DATA_BLOCK "DB3323"
TITLE =	TITLE ==CH2++ZNE02_Alarm_List
{ S7_language := '16(1) Italiano (Italia)  10.08.2015  13:02:09' }
VERSION : 0.1


  STRUCT
   CM_ID : STRING  [8 ] := '=CH2_2';	//IDENTIFICATIVO TRATTO
   STATION_ID : STRING  [8 ] := '++ZNE02';	//TRATTO - ZONA - STAZIONE
   ELEMENT_ID : STRING  [8 ];	//ELEMENTO
   DB_ID : INT  := 3;	//GRANDEZZA DB O TIPO
   PART_IDENTIFICATION : STRING  [12 ];	//IDENTIFICAZIONE PEZZO IN LAVORAZIONE
   ACT_CYCLE_TIME : INT ;	//TEMPO CICLO EFFETTIVO
   COUNT_GOOD : INT ;	//PEZZO PRODOTTO BUONO
   COUNT_SCRAP : INT ;	//PEZZO PRODOTTO DI SCARTO
   ACCUMULATORS : ARRAY  [0 .. 15 ] OF //ACCUMULI
   INT ;
   SPARE_01 : ARRAY  [0 .. 17 ] OF //RISERVE
   INT ;
   CODE_EVENT : ARRAY  [0 .. 7 ] OF //CODICI DI DIAGNOSTICA (codici a 4 cifre)
   INT ;
   EVENTS : STRUCT 	//EVENTI DI DIAGNOSTICA / MONITORAGGIO (bit)
    E0001 : BOOL ;	//=CH2_2++ZNE02+HCZ01-DMC01;FALHA NO MÓDULO ET200S;1
    E0002 : BOOL ;	//=CH2_2++ZNE02+HCZ01-DSW01;FALHA DE SCALANCE;1
    E0003 : BOOL ;	//=CH2_2++ZNE02+HCZ01-QF_06;ALIMENTAÇÃO MAGNETOTÉRMICA PARA CIRCUITOS AUXILIARES;1
    E0004 : BOOL ;	//=CH2_2++ZNE02+HCZ01-QF_07;POTÊNCIA MAGNETOTÉRMICA. COMANDOS E SINAIS DE SAÍDA;1
    E0005 : BOOL ;	//=CH2_2++ZNE02+HCZ01-QF_08;MAGNETOTHERM.;1
    E0006 : BOOL ;	//=CH2_2++ZNE02+HCZ01-QF_09;POTÊNCIA MAGNETOTÉRMICA. MÓDULOS E SWITCHES E/S ET200;1
    E0007 : BOOL ;
    E0008 : BOOL ;
    E0009 : BOOL ;	//=CH2_2++ZNE02+HKL02-SQ_04;MANIPULADORES DIREITOS COMPACTOS;1
    E0010 : BOOL ;	//=CH2_2++ZNE02+HKL02-SQ_10;MANIPULADORES ESQUERDOS EM TAMANHO COMPACTO;1
    E0011 : BOOL ;
    E0012 : BOOL ;
    E0013 : BOOL ;
    E0014 : BOOL ;
    E0015 : BOOL ;
    E0016 : BOOL ;
    E0017 : BOOL ;	//=CH2_2++ZNE02+HCZ01-QF_25;GRUPO DE ROTAÇÃO DA FONTE DE ALIMENTAÇÃO 440Vac +CR_01;1
    E0018 : BOOL ;	//=CH2_2++ZNE02+HCZ01-QF_26;PODER GRUPO DE ROTAÇÃO DE BACKUP 440Vac +CR_01;1
    E0019 : BOOL ;	//=CH2_2++ZNE02+HCZ01-QF_27;GRUPO DE ROTAÇÃO DA FONTE DE ALIMENTAÇÃO 440Vac +CR_02;1
    E0020 : BOOL ;	//=CH2_2++ZNE02+HCZ01-QF_28;PODER GRUPO DE ROTAÇÃO DE BACKUP 440Vac +CR_02;1
    E0021 : BOOL ;	//=CH2_2++ZNE02+HCZ01-QF_29;FONTE DE ALIMENTAÇÃO 440Vac CADEIA+TC_01;1
    E0022 : BOOL ;	//=CH2_2++ZNE02+HCZ01-QF_30;MAGNETOTHERM.440Vac FREIO GR.ROTAÇÃO +CR_01;1
    E0023 : BOOL ;	//=CH2_2++ZNE02+HCZ01-QF_31;MAGNETOTHERM.440Vac FREIO GR.ROTAÇÃO BK +CR_01;1
    E0024 : BOOL ;	//=CH2_2++ZNE02+HCZ01-QF_32;MAGNETOTHERM.440Vac FREIO GR.ROTAÇÃO +CR_02;1
    E0025 : BOOL ;	//=CH2_2++ZNE02+HCZ01-QF_33;MAGNETOTHERM.440Vac FREIO GR.ROTAÇÃO BK +CR_02;1
    E0026 : BOOL ;	//=CH2_2++ZNE02+HCZ01-QF_34;MAGNETOTERM.440Vac FREIO DE CORRENTE +TC_01;1
    E0027 : BOOL ;	//=CH2_2++ZNE02+HCZ01-QF_35;MAGNETOTERM.440Vac CADEIA DE BACKUP +TC_01;1
    E0028 : BOOL ;	//=CH2_2++ZNE02+HCZ01-QF_36;MAGNETOTERM.440Vac FREIO DE CORRENTE DE BACKUP +TC_01;1
    E0029 : BOOL ;	//=CH2_2++ZNE02+HCZ01-BT_01;SOBRETEMPERATURA DO RESISTOR DE FRENAGEM +CR_01;1
    E0030 : BOOL ;	//=CH2_2++ZNE02+HCZ01-BT_02;SOBRETEMP DO RESISTOR DE FRENAGEM DE BACKUP.;1
    E0031 : BOOL ;	//=CH2_2++ZNE02+HCZ01-BT_03;SOBRETEMPERATURA DO RESISTOR DE FRENAGEM +CR_02;1
    E0032 : BOOL ;	//=CH2_2++ZNE02+HCZ01-BT_04;SOBRETEMP DO RESISTOR DE FRENAGEM DE BACKUP.;1
    E0033 : BOOL ;	//=CH2_2++ZNE02+HCZ01-U__01;FALHA MOVIDRIVE +CR_01;1
    E0034 : BOOL ;	//=CH2_2++ZNE02+HCZ01-U__02;FALHA DE BACKUP DO MOVIDRIVE +CR_01;1
    E0035 : BOOL ;	//=CH2_2++ZNE02+HCZ01-U__03;FALHA MOVIDRIVE +CR_02;1
    E0036 : BOOL ;	//=CH2_2++ZNE02+HCZ01-U__04;FALHA DE BACKUP DO MOVIDRIVE +CR_02;1
    E0037 : BOOL ;	//=CH2_2++ZNE02+HCZ01-U__05;FALHA MOVIDRIVE +TC_01;1
    E0038 : BOOL ;	//=CH2_2++ZNE02+HCZ01-U__06;FALHA DE BACKUP DO MOVIDRIVE +TC_01;1
    E0039 : BOOL ;	//=CH2_2++ZNE02+HCZ01-U__01;MOVIDRIVE +CR_01 ERRO DE COMUNICAÇÃO;1
    E0040 : BOOL ;	//=CH2_2++ZNE02+HCZ01-U__02;ERRO DE COMUNICAÇÃO BACKUP DO MOVIDRIVE +CR_01;1
    E0041 : BOOL ;	//=CH2_2++ZNE02+HCZ01-U__03;MOVIDRIVE +CR_02 ERRO DE COMUNICAÇÃO;1
    E0042 : BOOL ;	//=CH2_2++ZNE02+HCZ01-U__04;ERRO DE COMUNICAÇÃO BACKUP DO MOVIDRIVE +CR_02;1
    E0043 : BOOL ;	//=CH2_2++ZNE02+HCZ01-U__05;MOVIDRIVE +TC_01 ERRO DE COMUNICAÇÃO;1
    E0044 : BOOL ;	//=CH2_2++ZNE02+HCZ01-U__06;ERRO COMUNICADO. BACKUP DO MOVIDRIVE +TC_01;1
    E0045 : BOOL ;	//=CH2_2++ZNE02+HCZ01-KMS02;EFICIÊNCIA DO RELÉ 440Vac SET_2 +CR_01;1
    E0046 : BOOL ;	//=CH2_2++ZNE02+HCZ01-KMS04;EFICIÊNCIA DO RELÉ 440Vca SET_4 +CR_02;1
    E0047 : BOOL ;	//=CH2_2++ZNE02+HCZ01-KMS06;EFICIÊNCIA DO RELÉ 440Vac SET_5 +TC_01;1
    E0048 : BOOL ;	//=CH2_2++ZNE02+HCZ01-KAS02;CONJUNTO DE EFICIÊNCIA DO RELÉ 24Vdc_2 +CR_01;1
    E0049 : BOOL ;	//=CH2_2++ZNE02+HCZ01-KAS04;CONJUNTO DE EFICIÊNCIA DO RELÉ 24Vdc_4 +CR_02;1
    E0050 : BOOL ;	//=CH2_2++ZNE02+HCZ01-KAS06;CONJUNTO DE EFICIÊNCIA DO RELÉ 24Vdc_5 +TC_01;1
    E0051 : BOOL ;	//=CH2_2++ZNE02+PTZ01-DMC01;FALHA NO MÓDULO ET200S;1
    E0052 : BOOL ;	//=CH2_2++ZNE02+PTZ02-DMC01;FALHA NO MÓDULO ET200S;1
    E0053 : BOOL ;	//=CH2_2++ZNE02+HKL01-DMC01;FALHA NO MÓDULO ET200S;1
    E0054 : BOOL ;	//=CH2_2++ZNE02+HKL02-DMC01;FALHA NO MÓDULO ET200S;1
    E0055 : BOOL ;	//=CH2_2++ZNE02+XGA01-SC_01;PORTÃO EM ANOMALIA;1
    E0056 : BOOL ;	//=CH2_2++ZNE02+XGA02-SC_01;PORTÃO EM ANOMALIA;1
    E0057 : BOOL ;	//=CH2_2++ZNE02+XGA05-SC_01;PORTÃO EM ANOMALIA;1
    E0058 : BOOL ;	//=CH2_2++ZNE02+XGA06-SC_01;PORTÃO EM ANOMALIA;1
    E0059 : BOOL ;
    E0060 : BOOL ;
    E0061 : BOOL ;
    E0062 : BOOL ;
    E0063 : BOOL ;
    E0064 : BOOL ;
    E0065 : BOOL ;	//=CH2_2++ZNE02+HCZ01-DMC01;ANOMALIA DO MÓDULO ProfSafe ET200S-FDI-FDO;2
    E0066 : BOOL ;	//=CH2_2++ZNE02+PTZ01-DMC01;ANOMALIA DO MÓDULO ProfSafe ET200S-FDI;2
    E0067 : BOOL ;	//=CH2_2++ZNE02+PTZ02-DMC01;ANOMALIA DO MÓDULO ProfSafe ET200S-FDI;2
    E0068 : BOOL ;	//=CH2_2++ZNE02+PTZ03-DMC01;ANOMALIA DO MÓDULO ProfSafe ET200S-FDI;2
    E0069 : BOOL ;	//=CH2_2++ZNE02+PRE01-DMC01;ANOMALIA DO MÓDULO ProfSafe ET200S-FDI;2
    E0070 : BOOL ;	//=CH2_2++ZNE02+HKL01-DMC01;ANOMALIA DO MÓDULO ProfSafe ET200S-FDI;2
    E0071 : BOOL ;	//=CH2_2++ZNE02+HKL02-DMC01;ANOMALIA DO MÓDULO ProfSafe ET200S-FDI;2
    E0072 : BOOL ;
    E0073 : BOOL ;
    E0074 : BOOL ;
    E0075 : BOOL ;
    E0076 : BOOL ;
    E0077 : BOOL ;	//=CH2_2++ZNE02+XGA06-SC_01;MANUTENÇÃO PROGRAMADA DE ACESSO ABERTO (PM);13
    E0078 : BOOL ;	//=CH2_2++ZNE02+XGA06-SC_01;LIMPEZA TÉCNICA DE ACESSO ABERTO (AM);14
    E0079 : BOOL ;	//=CH2_2++ZNE02+XGA06-SC_01;ACESSO NÃO RESTAURADO MANUTENÇÃO DO PROGRAMA (PM);13
    E0080 : BOOL ;	//=CH2_2++ZNE02+XGA06-SC_01;ACESSO NÃO RESTAURADO LIMPEZA TÉCNICA (AM);14
    E0081 : BOOL ;	//=CH2_2++ZNE02+PTZ01-SB_07;BOTÃO DE EMERGENCIA APERTADO;2
    E0082 : BOOL ;	//=CH2_2++ZNE02+PTZ01-SB_07;EMERGÊNCIA NÃO RESTAURADA;2
    E0083 : BOOL ;	//=CH2_2++ZNE02+PTZ02-SB_07;BOTÃO DE EMERGENCIA APERTADO;2
    E0084 : BOOL ;	//=CH2_2++ZNE02+PTZ02-SB_07;EMERGÊNCIA NÃO RESTAURADA;2
    E0085 : BOOL ;	//=CH2_2++ZNE02+PGA01-SB_01;BOTÃO DE EMERGENCIA APERTADO;2
    E0086 : BOOL ;	//=CH2_2++ZNE02+PGA01-SB_01;EMERGÊNCIA NÃO RESTAURADA;2
    E0087 : BOOL ;	//=CH2_2++ZNE02+PGA02-SB_01;BOTÃO DE EMERGENCIA APERTADO;2
    E0088 : BOOL ;	//=CH2_2++ZNE02+PGA02-SB_01;EMERGÊNCIA NÃO RESTAURADA;2
    E0089 : BOOL ;	//=CH2_2++ZNE02+SLL01-SB_01;CORDA DE EMERGÊNCIA DO LADO ESQUERDO PUXADA;2
    E0090 : BOOL ;	//=CH2_2++ZNE02+SLL01-SB_01;CORDA DE EMERGÊNCIA LADO ESQUERDO NÃO RESTAURADA;2
    E0091 : BOOL ;	//=CH2_2++ZNE02+SLL02-SB_01;CORDA DE EMERGÊNCIA DO LADO DIREITO PUXADA;2
    E0092 : BOOL ;	//=CH2_2++ZNE02+SLL02-SB_01;CORDA DE EMERGÊNCIA LADO DIREITO NÃO RESTAURADA;2
    E0093 : BOOL ;	//=CH2_2++ZNE02+SLL03-SB_01;CORDA DE EMERGÊNCIA DO LADO ESQUERDO PUXADA;2
    E0094 : BOOL ;	//=CH2_2++ZNE02+SLL03-SB_01;CORDA DE EMERGÊNCIA LADO ESQUERDO NÃO RESTAURADA;2
    E0095 : BOOL ;	//=CH2_2++ZNE02+SLL04-SB_01;CORDA DE EMERGÊNCIA DO LADO DIREITO PUXADA;2
    E0096 : BOOL ;	//=CH2_2++ZNE02+SLL04-SB_01;CORDA DE EMERGÊNCIA LADO DIREITO NÃO RESTAURADA;2
    E0097 : BOOL ;	//=CH2_2++ZNE02+SLL05-SB_01;CORDA DE EMERGÊNCIA DO LADO ESQUERDO PUXADA;2
    E0098 : BOOL ;	//=CH2_2++ZNE02+SLL05-SB_01;CORDA DE EMERGÊNCIA LADO ESQUERDO NÃO RESTAURADA;2
    E0099 : BOOL ;	//=CH2_2++ZNE02+SLL06-SB_01;CORDA DE EMERGÊNCIA DO LADO DIREITO PUXADA;2
    E0100 : BOOL ;	//=CH2_2++ZNE02+SLL06-SB_01;CORDA DE EMERGÊNCIA LADO DIREITO NÃO RESTAURADA;2
    E0101 : BOOL ;	//=CH2_2++ZNE02+XGA01-SC_01;ACESSO ABERTO NÃO PROGRAMADO (GM);2
    E0102 : BOOL ;	//=CH2_2++ZNE02+XGA01-SC_01;ACESSO NÃO RESTAURADO(GM);2
    E0103 : BOOL ;	//=CH2_2++ZNE02+XGA02-SC_01;ACESSO ABERTO NÃO PROGRAMADO (GM);2
    E0104 : BOOL ;	//=CH2_2++ZNE02+XGA02-SC_01;ACESSO NÃO RESTAURADO(GM);2
    E0105 : BOOL ;	//=CH2_2++ZNE02+XGA05-SC_01;ACESSO ABERTO NÃO PROGRAMADO (GM);2
    E0106 : BOOL ;	//=CH2_2++ZNE02+XGA05-SC_01;ACESSO NÃO RESTAURADO(GM);2
    E0107 : BOOL ;	//=CH2_2++ZNE02+XGA06-SC_01;ACESSO ABERTO NÃO PROGRAMADO (GM);2
    E0108 : BOOL ;	//=CH2_2++ZNE02+XGA06-SC_01;ACESSO NÃO RESTAURADO(GM);2
    E0109 : BOOL ;	//=CH2_2++ZNE02+PRB01-VT_01;BARREIRA ATIVADA (ESTAÇÃO 77);2
    E0110 : BOOL ;	//=CH2_2++ZNE02+PRB01-VT_01;BARREIRA NÃO RESTAURADA (ESTAÇÃO 77);2
    E0111 : BOOL ;	//=CH2_2++ZNE02+PRB02-VT_02;BARREIRA ATIVADA (ESTAÇÃO 78);2
    E0112 : BOOL ;	//=CH2_2++ZNE02+PRB02-VT_02;BARREIRA NÃO RESTAURADA (ESTAÇÃO 78);2
    E0113 : BOOL ;	//=CH2_2++ZNE02+PRB03-VT_03;BARREIRA ATIVADA (ESTAÇÃO Q2);2
    E0114 : BOOL ;	//=CH2_2++ZNE02+PRB03-VT_03;BARREIRA NÃO RESTAURADA (ESTAÇÃO Q2);2
    E0115 : BOOL ;	//=CH2_2++ZNE02+PRB04-VT_04;BARREIRA ATIVADA (ESTAÇÃO Q3);2
    E0116 : BOOL ;	//=CH2_2++ZNE02+PRB04-VT_04;BARREIRA NÃO RESTAURADA (ESTAÇÃO Q3);2
    E0117 : BOOL ;	//=CH2_2++ZNE02+XGA01-SC_01;MANUTENÇÃO PROGRAMADA DE ACESSO ABERTO (PM);13
    E0118 : BOOL ;	//=CH2_2++ZNE02+XGA01-SC_01;LIMPEZA TÉCNICA DE ACESSO ABERTO (AM);14
    E0119 : BOOL ;	//=CH2_2++ZNE02+XGA01-SC_01;ACESSO NÃO RESTAURADO PROG. DE MANUTENÇÃO (PM);13
    E0120 : BOOL ;	//=CH2_2++ZNE02+XGA01-SC_01;ACESSO NÃO RESTAURADO LIMPEZA TÉCNICA (AM);14
    E0121 : BOOL ;	//=CH2_2++ZNE02+XGA02-SC_01;MANUTENÇÃO PROGRAMADA DE ACESSO ABERTO (PM);13
    E0122 : BOOL ;	//=CH2_2++ZNE02+XGA02-SC_01;LIMPEZA TÉCNICA DE ACESSO ABERTO (AM);14
    E0123 : BOOL ;	//=CH2_2++ZNE02+XGA02-SC_01;ACESSO NÃO RESTAURADO PROG. DE MANUTENÇÃO (PM);13
    E0124 : BOOL ;	//=CH2_2++ZNE02+XGA02-SC_01;ACESSO NÃO RESTAURADO LIMPEZA TÉCNICA (AM);14
    E0125 : BOOL ;	//=CH2_2++ZNE02+XGA05-SC_01;MANUTENÇÃO PROGRAMADA DE ACESSO ABERTO (PM);13
    E0126 : BOOL ;	//=CH2_2++ZNE02+XGA05-SC_01;LIMPEZA TÉCNICA DE ACESSO ABERTO (AM);14
    E0127 : BOOL ;	//=CH2_2++ZNE02+XGA05-SC_01;ACESSO NÃO RESTAURADO PROG. DE MANUTENÇÃO (PM);13
    E0128 : BOOL ;	//=CH2_2++ZNE02+XGA05-SC_01;ACESSO NÃO RESTAURADO LIMPEZA TÉCNICA (AM);14
    E0129 : BOOL ;	//=CH2_2++ZNE02+HCZ01-QF_03;FONTE DE ALIMENTAÇÃO MAGNETOTÉRMICA PARA AR CONDICIONADO 400V;58
    E0130 : BOOL ;	//=CH2_2++ZNE02+HCZ01-QF_15;MAGNETO. PODER PAINEL OPERADOR 24Vdc +PTZ01;58
    E0131 : BOOL ;	//=CH2_2++ZNE02+HCZ01-QF_16;MAGNETO. PODER PAINEL OPERADOR 24Vdc +PTZ02;58
    E0132 : BOOL ;	//=CH2_2++ZNE02+HCZ01-U__01;PRÉ-ALARME MOVIDRIVE +CR_01;58
    E0133 : BOOL ;	//=CH2_2++ZNE02+HCZ01-U__02;PRÉ-ALARME DE BACKUP DO MOVIDRIVE +CR_01;58
    E0134 : BOOL ;	//=CH2_2++ZNE02+HCZ01-U__03;PRÉ-ALARME MOVIDRIVE +CR_02;58
    E0135 : BOOL ;	//=CH2_2++ZNE02+HCZ01-U__04;PRÉ-ALARME DE BACKUP DO MOVIDRIVE +CR_02;58
    E0136 : BOOL ;	//=CH2_2++ZNE02+HCZ01-U__05;PRÉ-ALARME MOVIDRIVE +TC_01;58
    E0137 : BOOL ;	//=CH2_2++ZNE02+HCZ01-U__06;PRÉ-ALARME DE BACKUP DO MOVIDRIVE +TC_01;58
    E0138 : BOOL ;	//=CH2_2++ZNE02+PTZ01-DSP01;PRÉ-ALARME SEM PLC <-> COMUNICAÇÃO IHM;58
    E0139 : BOOL ;	//=CH2_2++ZNE02+PTZ02-DSP01;PRÉ-ALARME SEM PLC <-> COMUNICAÇÃO IHM;58
    E0140 : BOOL ;	//=CH2_2++ZNE02+PTZ01-SA_03;PEDIDO DE ACESSO PARA MANUTENÇÃO PLANEJADA (PM);58
    E0141 : BOOL ;	//=CH2_2++ZNE02+PTZ01-SA_03;SOLICITAR ACESSO PARA LIMPEZA TÉCNICA (AM);58
    E0142 : BOOL ;	//=CH2_2++ZNE02+PTZ02-SA_03;PEDIDO DE ACESSO PARA MANUTENÇÃO PLANEJADA (PM);58
    E0143 : BOOL ;	//=CH2_2++ZNE02+PTZ02-SA_03;SOLICITAR ACESSO PARA LIMPEZA TÉCNICA (AM);58
    E0144 : BOOL ;	//=CH2_2++ZNE02+PGA01-SA_01;PEDIDO DE ACESSO PARA MANUTENÇÃO PLANEJADA (PM);58
    E0145 : BOOL ;	//=CH2_2++ZNE02+PGA01-SA_01;SOLICITAR ACESSO PARA LIMPEZA TÉCNICA (AM);58
    E0146 : BOOL ;	//=CH2_2++ZNE02+PGA02-SA_01;PEDIDO DE ACESSO PARA MANUTENÇÃO PLANEJADA (PM);58
    E0147 : BOOL ;	//=CH2_2++ZNE02+PGA02-SA_01;SOLICITAR ACESSO PARA LIMPEZA TÉCNICA (AM);58
    E0148 : BOOL ;	//=CH2_2++ZNE02+PTZ01-SA_03;SOLICITAR ACESSO PARA MANUTENÇÃO NÃO PROGRAMADA (GM);58
    E0149 : BOOL ;	//=CH2_2++ZNE02+PTZ02-SA_03;SOLICITAR ACESSO PARA MANUTENÇÃO NÃO PROGRAMADA (GM);58
    E0150 : BOOL ;	//=CH2_2++ZNE02+PGA01-SA_01;SOLICITAR ACESSO PARA MANUTENÇÃO NÃO PROGRAMADA (GM);58
    E0151 : BOOL ;	//=CH2_2++ZNE02+PGA02-SA_01;SOLICITAR ACESSO PARA MANUTENÇÃO NÃO PROGRAMADA (GM);58
    E0152 : BOOL ;	//=CH2_2++ZNE02+HCZ01-ST_01;CONTROLE DE TEMPERATURA DO GABINETE;58
    E0153 : BOOL ;	//=CH2_2++ZNE02+HAU01-QF_01;ALIMENTAÇÃO TÉRMICA 440Vac USUÁRIOS NO LADO DA LINHA;58
    E0154 : BOOL ;	//=CH2_2++ZNE02+HAU01-QF_02;PARAFUSO 220Vac TORX T50 PARA FIXAÇÃO. FIVELA DIREITA;58
    E0155 : BOOL ;	//=CH2_2++ZNE02+HAU01-QF_03;PARAFUSO FIXO TÉRMICO 220Vac. BANCO TRASEIRO =CH2++ZNE0;58
    E0156 : BOOL ;	//=CH2_2++ZNE02+HAU01-QF_04;ESTRUTURA TÉRMICA 220Vac FIX INFERIOR DIREITA =CH2++ZNE;58
    E0157 : BOOL ;	//=CH2_2++ZNE02+HAU01-QF_05;ÂNCORA/TUBO 220Vac. ESCAPE =CH2++ZNE02+FRM;58
    E0158 : BOOL ;	//=CH2_2++ZNE02+HAU01-QF_06;220Vac TORX T50 PARA FIXAÇÃO DE FILIAL ESQUERDO FIVELA =CH2++ZNE;58
    E0159 : BOOL ;	//=CH2_2++ZNE02+HAU01-QF_07;220Vac FIX SUPORTE INFERIOR ESQUERDO =CH2++ZNE02+FRM06;58
    E0160 : BOOL ;	//=CH2_2++ZNE02+HAU01-QF_08;ALIMENTAÇÃO TÉRMICA 220Vac USUÁRIO 7;58
    E0161 : BOOL ;	//=CH2_2++ZNE02+HAU01-QF_09;ALIMENTAÇÃO TÉRMICA 220Vac USUÁRIO 8;58
    E0162 : BOOL ;	//=CH2_2++ZNE02+HAU01-QF_10;ALIMENTAÇÃO TÉRMICA 220Vac USUÁRIO 9;58
    E0163 : BOOL ;	//=CH2_2++ZNE02+HCZ01;PRÉ-ALARME DE SEGURANÇA DE BYPASS ATIVO;54
    E0164 : BOOL ;
    E0165 : BOOL ;
    E0166 : BOOL ;
    E0167 : BOOL ;
    E0168 : BOOL ;
    E0169 : BOOL ;	//=CH2_2++ZNE02+HAU02-QF_01;ALIMENTAÇÃO TÉRMICA 440Vac USUÁRIOS NO LADO DA LINHA;58
    E0170 : BOOL ;	//=CH2_2++ZNE02+HAU02-QF_02;CRISTAIS 220Vac (CARGA) =CH2++ZNE02+PTN01;58
    E0171 : BOOL ;	//=CH2_2++ZNE02+HAU02-QF_03;PÁRA-BRISA 220Vac B.U - LINHA =CH2++ZNE02+FRM04;58
    E0172 : BOOL ;	//=CH2_2++ZNE02+HAU02-QF_04;ALIMENTAÇÃO TÉRMICA 220Vac USUÁRIO 3;58
    E0173 : BOOL ;	//=CH2_2++ZNE02+HAU02-QF_05;ALIMENTAÇÃO TÉRMICA 220Vac USUÁRIO 4;58
    E0174 : BOOL ;	//=CH2_2++ZNE02+HAU02-QF_06;ALIMENTAÇÃO TÉRMICA 220Vac USUÁRIO 5;58
    E0175 : BOOL ;	//=CH2_2++ZNE02+HAU02-QF_07;ALIMENTAÇÃO TÉRMICA 220Vac USUÁRIO 6;58
    E0176 : BOOL ;	//=CH2_2++ZNE02+HAU02-QF_08;ALIMENTAÇÃO TÉRMICA 220Vac USUÁRIO 7;58
    E0177 : BOOL ;	//=CH2_2++ZNE02+HAU02-QF_09;ALIMENTAÇÃO TÉRMICA 220Vac USUÁRIO 8;58
    E0178 : BOOL ;	//=CH2_2++ZNE02+HAU02-QF_10;ALIMENTAÇÃO TÉRMICA 220Vac USUÁRIO 9;58
    E0179 : BOOL ;
    E0180 : BOOL ;
    E0181 : BOOL ;
    E0182 : BOOL ;
    E0183 : BOOL ;
    E0184 : BOOL ;
    E0185 : BOOL ;	//=CH2_2++ZNE02+HAU03-QF_01;ALIMENTAÇÃO TÉRMICA 440Vac USUÁRIOS NO LADO DA LINHA;58
    E0186 : BOOL ;	//=CH2_2++ZNE02+HAU03-QF_02;ALIMENTAÇÃO TÉRMICA 220Vac USUÁRIO 1;58
    E0187 : BOOL ;	//=CH2_2++ZNE02+HAU03-QF_03;ALIMENTAÇÃO TÉRMICA 220Vac USUÁRIO 2;58
    E0188 : BOOL ;	//=CH2_2++ZNE02+HAU03-QF_04;ALIMENTAÇÃO TÉRMICA 220Vac USUÁRIO 3;58
    E0189 : BOOL ;	//=CH2_2++ZNE02+HAU03-QF_05;ALIMENTAÇÃO TÉRMICA 220Vac USUÁRIO 4;58
    E0190 : BOOL ;	//=CH2_2++ZNE02+HAU03-QF_06;ALIMENTAÇÃO TÉRMICA 220Vac USUÁRIO 5;58
    E0191 : BOOL ;	//=CH2_2++ZNE02+HAU03-QF_07;ALIMENTAÇÃO TÉRMICA 220Vac USUÁRIO 6;58
    E0192 : BOOL ;	//=CH2_2++ZNE02+HAU03-QF_08;ALIMENTAÇÃO TÉRMICA 220Vac USUÁRIO 7;58
    E0193 : BOOL ;	//=CH2_2++ZNE02+HAU03-QF_09;ALIMENTAÇÃO TÉRMICA 220Vac USUÁRIO 8;58
    E0194 : BOOL ;	//=CH2_2++ZNE02+HAU03-QF_10;ALIMENTAÇÃO TÉRMICA 220Vac USUÁRIO 9;58
    E0195 : BOOL ;
    E0196 : BOOL ;
    E0197 : BOOL ;
    E0198 : BOOL ;
    E0199 : BOOL ;
    E0200 : BOOL ;
    E0201 : BOOL ;	//=CH2_2++ZNE02+PTZ01;SETOR ASCENTE NÃO ESTÁ EM CICLO INICIADO;58
    E0202 : BOOL ;	//=CH2_2++ZNE02+PTZ01;SETOR JUSANTE NÃO ESTÁ EM CICLO INICIADO;58
    E0203 : BOOL ;	//=CH2_2++ZNE02+PTZ02;SETOR ASCENTE NÃO ESTÁ EM CICLO INICIADO;58
    E0204 : BOOL ;	//=CH2_2++ZNE02+PTZ02;SETOR JUSANTE NÃO ESTÁ EM CICLO INICIADO;58
    E0205 : BOOL ;	//=CH2_2++ZNE02+PTZ03;SETOR ASCENTE NÃO ESTÁ EM CICLO INICIADO;58
    E0206 : BOOL ;	//=CH2_2++ZNE02+PTZ03;SETOR JUSANTE NÃO ESTÁ EM CICLO INICIADO;58
    E0207 : BOOL ;	//=CH2_2++ZNE02+PRE01;SETOR ASCENTE NÃO ESTÁ EM CICLO INICIADO;58
    E0208 : BOOL ;	//=CH2_2++ZNE02+PRE01;SETOR JUSANTE NÃO ESTÁ EM CICLO INICIADO;58
    E0209 : BOOL ;	//=CH2_2++ZNE02;EM PRODUÇÃO;19
    E0210 : BOOL ;	//=CH2_2++ZNE02+PTZ01-SB_05;INICIAR CICLO AUTOMÁTICO;15
    E0211 : BOOL ;	//=CH2_2++ZNE02+PTZ02-SB_05;INICIAR CICLO AUTOMÁTICO;15
    E0212 : BOOL ;	//=CH2_2++ZNE02+PTZ01-SA_01;CICLO MANUAL SELECIONADO;16
    E0213 : BOOL ;	//=CH2_2++ZNE02+PTZ02-SA_01;CICLO MANUAL SELECIONADO;16
    E0214 : BOOL ;	//=CH2_2++ZNE02+PTZ01-SB_04;PARADA DO CICLO;17
    E0215 : BOOL ;	//=CH2_2++ZNE02+PTZ02-SB_04;PARADA DO CICLO;17
    E0216 : BOOL ;
    E0217 : BOOL ;
    E0218 : BOOL ;
    E0219 : BOOL ;
    E0220 : BOOL ;
    E0221 : BOOL ;
    E0222 : BOOL ;
    E0223 : BOOL ;
    E0224 : BOOL ;
    E0225 : BOOL ;	//=CH2_2++ZNE02+TC_01-SQ_04;FC FALHA DENTE PARADA TEMPORÁRIA SEM GANCHO;1
    E0226 : BOOL ;	//=CH2_2++ZNE02+TC_01-SQ_05;FC FALHA DENTE PARADA TEMPORÁRIA SEM GANCHO;1
    E0227 : BOOL ;
    E0228 : BOOL ;
    E0229 : BOOL ;
    E0230 : BOOL ;	//=CH2_2++ZNE02+TC_01-SQ_06;CONTROLE ANTI-VARA DE CADEIA;1
    E0231 : BOOL ;
    E0232 : BOOL ;
    E0233 : BOOL ;	//=CH2_2++ZNE02+TC_01-SE_01;CONTROLE DE ROTAÇÃO DA CADEIA;1
    E0234 : BOOL ;	//=CH2_2++ZNE02+TC_01-B__01;VERIFICAÇÃO DE CADEIA LENTA;1
    E0235 : BOOL ;	//=CH2_2++ZNE02+TC_01-SE_01;FALHA DO CODIFICADOR WIP;1
    E0236 : BOOL ;
    E0237 : BOOL ;	//=CH2_2++ZNE02+TC_01;CTRL EXECUTAR TTS ENTRADA DO CHASSIS;1
    E0238 : BOOL ;	//=CH2_2++ZNE02+TC_01;CTRL RUN TTS SAÍDA DO CHASSIS;1
    E0239 : BOOL ;
    E0240 : BOOL ;
    E0241 : BOOL ;	//=CH2_2++ZNE02+TC_01;PARCEIRO 1 NÃO FORA DO LADO ESQUERDO;10
    E0242 : BOOL ;	//=CH2_2++ZNE02+TC_01;PARCEIRO 2 NÃO FORA DAS DIMENSÕES DO LADO DIREITO;10
    E0243 : BOOL ;	//=CH2_2++ZNE02+TC_01;PARCEIRO 3 NÃO FORA DO LADO ESQUERDO;10
    E0244 : BOOL ;	//=CH2_2++ZNE02+TC_01;PARCEIRO 4 NÃO FORA DAS DIMENSÕES DO LADO DIREITO;10
    E0245 : BOOL ;	//=CH2_2++ZNE02+TC_01;PARCEIRO 5 NÃO FORA DO LADO ESQUERDO;10
    E0246 : BOOL ;	//=CH2_2++ZNE02+TC_01;PARCEIRO 6 NÃO FORA DAS DIMENSÕES DO LADO DIREITO;10
    E0247 : BOOL ;	//=CH2_2++ZNE02+TC_01;PARCEIRO 7 NÃO FORA DO LADO ESQUERDO;10
    E0248 : BOOL ;	//=CH2_2++ZNE02+TC_01;PARCEIRO 8 NÃO FORA DAS DIMENSÕES DO LADO DIREITO;10
    E0249 : BOOL ;	//=CH2_2++ZNE02+TC_01;PRÉ-ALARME DE BYPASS DE FALHA ATIVO;58
    E0250 : BOOL ;	//=CH2_2++ZNE02+TC_01;FALTA PRÉ-ALARME DE HABILITAÇÃO MECÂNICA;58
    E0251 : BOOL ;
    E0252 : BOOL ;
    E0253 : BOOL ;
    E0254 : BOOL ;
    E0255 : BOOL ;
    E0256 : BOOL ;
    E0257 : BOOL ;	//=CH2_2++ZNE02+TC_01;FALHA NO CARREGAMENTO;6
    E0258 : BOOL ;	//=CH2_2++ZNE02+TC_01;FALHA NO DESCARREGAMENTO;9
    E0259 : BOOL ;
    E0260 : BOOL ;
    E0261 : BOOL ;
    E0262 : BOOL ;
    E0263 : BOOL ;
    E0264 : BOOL ;
    E0265 : BOOL ;	//=CH2_2++ZNE02+TC_01;ESVAZIAMENTO EM ANDAMENTO;58
    E0266 : BOOL ;
    E0267 : BOOL ;
    E0268 : BOOL ;
    E0269 : BOOL ;
    E0270 : BOOL ;
    E0271 : BOOL ;
    E0272 : BOOL ;
    E0273 : BOOL ;	//=CH2_2++ZNE02+CR_01-SQ_01;VERIFIQUE A QUEBRA DA CORRENTE DIREITA;1
    E0274 : BOOL ;	//=CH2_2++ZNE02+CR_01-SQ_02;VERIFIQUE A QUEBRA DA CORRENTE ESQUERDA;1
    E0275 : BOOL ;	//=CH2_2++ZNE02+CR_01-SQ_03;VERIFICAÇÃO DO BLOCO DE SEGURANÇA DO GANCHO DE FALHA FC;1
    E0276 : BOOL ;
    E0277 : BOOL ;	//=CH2_2++ZNE02+CR_01-SQ_05;CONTROLE DE POSIÇÃO DE REPOUSO DE FALHA FC;1
    E0278 : BOOL ;	//=CH2_2++ZNE02+CR_01-SQ_06;Obturador desengatado;1
    E0279 : BOOL ;	//=CH2_2++ZNE02+CR_01-SQ_07;FC FALHA INÍCIO DE ROTAÇÃO DO GANCHO;1
    E0280 : BOOL ;	//=CH2_2++ZNE02+CR_01-SQ_08;CONTROLE DE POSIÇÃO DE FALHA FC NO TRABALHO;1
    E0281 : BOOL ;	//=CH2_2++ZNE02+CR_01-SQ_09;FALHA DO FC FORA DO ESPAÇO;1
    E0282 : BOOL ;	//=CH2_2++ZNE02+CR_01-SQE01;EXTRACURSO GR. ROTAÇÃO DE DESCANSO;1
    E0283 : BOOL ;	//=CH2_2++ZNE02+CR_01-SQE02;EXTRACURSO GR. ROTAÇÃO DE TRABALHO;1
    E0284 : BOOL ;	//=CH2_2++ZNE02+CR_01-SQA01;FC FALHA ROTAÇÃO DO GANCHO PARADA DESCANSO;1
    E0285 : BOOL ;	//=CH2_2++ZNE02+CR_01-SQA02;FC FAULT STOP TRABALHO DE ROTAÇÃO DO GANCHO;1
    E0286 : BOOL ;	//=CH2_2++ZNE02+CR_01-SQS01;FC FALHA ROTAÇÃO DO GANCHO LENTA;1
    E0287 : BOOL ;	//=CH2_2++ZNE02+CR_01-SQS02;FALHA FC DESACELERAÇÃO DA ROTAÇÃO DO GANCHO DE TRABALHO;1
    E0288 : BOOL ;	//=CH2_2++ZNE02+CR_01-SQ_10;FC FALHA PRESENÇA DA RODA CAM DO OBTURADOR;1
    E0289 : BOOL ;	//=CH2_2++ZNE02+CR_01-SQ_04;CONTROLE DE BLOQUEIO DE ROTAÇÃO;1
    E0290 : BOOL ;	//=CH2_2++ZNE02+CR_01-SQA01;TEMPO DE ROTAÇÃO DO GANCHO EM REPOUSO;1
    E0291 : BOOL ;	//=CH2_2++ZNE02+CR_01-SQA02;TEMPO DE ROTAÇÃO DO GANCHO NO TRABALHO;1
    E0292 : BOOL ;	//=CH2_2++ZNE02+CR_01;FORA DA ETAPA_00;1
    E0293 : BOOL ;	//=CH2_2++ZNE02+CR_01;FORA DA ETAPA_05;1
    E0294 : BOOL ;	//=CH2_2++ZNE02+CR_01;FORA DA ETAPA_10;1
    E0295 : BOOL ;	//=CH2_2++ZNE02+CR_01;FORA DA ETAPA_15;1
    E0296 : BOOL ;	//=CH2_2++ZNE02+CR_01;FALHA NA ROTAÇÃO DO GANCHO;1
    E0297 : BOOL ;	//=CH2_2++ZNE02+CR_01;ANOMALIA DE SELEÇÃO DE LINHA/BACKUP MOVIDRIVE;1
    E0298 : BOOL ;	//=CH2_2++ZNE02+CR_01-M__01;ALARME DE CORRENTE ABSORVIDA;1
    E0299 : BOOL ;
    E0300 : BOOL ;
    E0301 : BOOL ;
    E0302 : BOOL ;
    E0303 : BOOL ;
    E0304 : BOOL ;
    E0305 : BOOL ;	//=CH2_2++ZNE02+CR_01;PRÉ-ALARME DE CORRENTE SOLTA;58
    E0306 : BOOL ;
    E0307 : BOOL ;
    E0308 : BOOL ;
    E0309 : BOOL ;
    E0310 : BOOL ;
    E0311 : BOOL ;
    E0312 : BOOL ;
    E0313 : BOOL ;	//=CH2_2++ZNE02+CR_01;PRÉ-ALARME DE BYPASS DE FALHA ATIVO;58
    E0314 : BOOL ;
    E0315 : BOOL ;
    E0316 : BOOL ;
    E0317 : BOOL ;
    E0318 : BOOL ;
    E0319 : BOOL ;
    E0320 : BOOL ;
    E0321 : BOOL ;
    E0322 : BOOL ;
    E0323 : BOOL ;
    E0324 : BOOL ;
    E0325 : BOOL ;
    E0326 : BOOL ;
    E0327 : BOOL ;
    E0328 : BOOL ;
    E0329 : BOOL ;	//=CH2_2++ZNE02+CR_01;CICLO AUTOMÁTICO PASSO A PASSO INICIADO;58
    E0330 : BOOL ;
    E0331 : BOOL ;
    E0332 : BOOL ;
    E0333 : BOOL ;
    E0334 : BOOL ;
    E0335 : BOOL ;
    E0336 : BOOL ;
    E0337 : BOOL ;	//=CH2_2++ZNE02+CR_02-SQ_01;VERIFIQUE A QUEBRA DA CORRENTE DIREITA;1
    E0338 : BOOL ;	//=CH2_2++ZNE02+CR_02-SQ_02;VERIFIQUE A QUEBRA DA CORRENTE ESQUERDA;1
    E0339 : BOOL ;	//=CH2_2++ZNE02+CR_02-SQ_03;VERIFICAÇÃO DO BLOCO DE SEGURANÇA DO GANCHO DE FALHA FC;1
    E0340 : BOOL ;
    E0341 : BOOL ;	//=CH2_2++ZNE02+CR_02-SQ_05;CONTROLE DE POSIÇÃO DE REPOUSO DE FALHA FC;1
    E0342 : BOOL ;	//=CH2_2++ZNE02+CR_02-SQ_06;Obturador desengatado;1
    E0343 : BOOL ;	//=CH2_2++ZNE02+CR_02-SQ_07;FC FALHA INÍCIO DE ROTAÇÃO DO GANCHO;1
    E0344 : BOOL ;	//=CH2_2++ZNE02+CR_02-SQ_08;CONTROLE DE POSIÇÃO DE FALHA FC NO TRABALHO;1
    E0345 : BOOL ;	//=CH2_2++ZNE02+CR_02-SQ_09;FALHA DO FC FORA DO ESPAÇO;1
    E0346 : BOOL ;	//=CH2_2++ZNE02+CR_02-SQE01;EXTRACURSO GR. ROTAÇÃO DE DESCANSO;1
    E0347 : BOOL ;	//=CH2_2++ZNE02+CR_02-SQE02;EXTRACURSO GR. ROTAÇÃO DE TRABALHO;1
    E0348 : BOOL ;	//=CH2_2++ZNE02+CR_02-SQA01;FC FALHA ROTAÇÃO DO GANCHO PARADA DESCANSO;1
    E0349 : BOOL ;	//=CH2_2++ZNE02+CR_02-SQA02;FC FAULT STOP TRABALHO DE ROTAÇÃO DO GANCHO;1
    E0350 : BOOL ;	//=CH2_2++ZNE02+CR_02-SQS01;FC FALHA ROTAÇÃO DO GANCHO LENTA;1
    E0351 : BOOL ;	//=CH2_2++ZNE02+CR_02-SQS02;FALHA FC DESACELERAÇÃO DA ROTAÇÃO DO GANCHO DE TRABALHO;1
    E0352 : BOOL ;	//=CH2_2++ZNE02+CR_02-SQ_10;FC FALHA PRESENÇA DA RODA CAM DO OBTURADOR;1
    E0353 : BOOL ;	//=CH2_2++ZNE02+CR_02-SQ_04;CONTROLE DE BLOQUEIO DE ROTAÇÃO;1
    E0354 : BOOL ;	//=CH2_2++ZNE02+CR_02-SQA01;TEMPO DE ROTAÇÃO DO GANCHO EM REPOUSO;1
    E0355 : BOOL ;	//=CH2_2++ZNE02+CR_02-SQA02;TEMPO DE ROTAÇÃO DO GANCHO NO TRABALHO;1
    E0356 : BOOL ;	//=CH2_2++ZNE02+CR_02;FORA DA ETAPA_00;1
    E0357 : BOOL ;	//=CH2_2++ZNE02+CR_02;FORA DA ETAPA_05;1
    E0358 : BOOL ;	//=CH2_2++ZNE02+CR_02;FORA DA ETAPA_10;1
    E0359 : BOOL ;	//=CH2_2++ZNE02+CR_02;FORA DA ETAPA_15;1
    E0360 : BOOL ;	//=CH2_2++ZNE02+CR_02;FALHA NA ROTAÇÃO DO GANCHO;1
    E0361 : BOOL ;	//=CH2_2++ZNE02+CR_02;ANOMALIA DE SELEÇÃO DE LINHA/BACKUP MOVIDRIVE;1
    E0362 : BOOL ;	//=CH2_2++ZNE02+CR_02-M__01;ALARME DE CORRENTE ABSORVIDA;1
    E0363 : BOOL ;
    E0364 : BOOL ;
    E0365 : BOOL ;
    E0366 : BOOL ;
    E0367 : BOOL ;
    E0368 : BOOL ;
    E0369 : BOOL ;	//=CH2_2++ZNE02+CR_02;PRÉ-ALARME DE CORRENTE SOLTA;58
    E0370 : BOOL ;
    E0371 : BOOL ;
    E0372 : BOOL ;
    E0373 : BOOL ;
    E0374 : BOOL ;
    E0375 : BOOL ;
    E0376 : BOOL ;
    E0377 : BOOL ;	//=CH2_2++ZNE02+CR_02;PRÉ-ALARME DE BYPASS DE FALHA ATIVO;58
    E0378 : BOOL ;
    E0379 : BOOL ;
    E0380 : BOOL ;
    E0381 : BOOL ;
    E0382 : BOOL ;
    E0383 : BOOL ;
    E0384 : BOOL ;
    E0385 : BOOL ;
    E0386 : BOOL ;
    E0387 : BOOL ;
    E0388 : BOOL ;
    E0389 : BOOL ;
    E0390 : BOOL ;
    E0391 : BOOL ;
    E0392 : BOOL ;
    E0393 : BOOL ;	//=CH2_2++ZNE02+CR_02;CICLO AUTOMÁTICO PASSO A PASSO INICIADO;58
    E0394 : BOOL ;	//=CH2_2++ZNE02+WIP01;Anomalia na leitura de código de barras/etiqueta;5
    E0395 : BOOL ;	//=CH2_2++ZNE02+WIP01;Tempo limite de leitura de código de barras/etiqueta;5
    E0396 : BOOL ;	//=CH2_2++ZNE02+WIP01;Inconsistência físico-lógica;5
    E0397 : BOOL ;	//=CH2_2++ZNE02+WIP01;Dígito de verificação CIS incorreto;5
    E0398 : BOOL ;	//=CH2_2++ZNE02+WIP01;Tempo limite de recepção de dados da rota anterior;5
    E0399 : BOOL ;	//=CH2_2++ZNE02+WIP01;Inconsistência de dados do ponto de ajuste do CIS/VIS com o CIS/VIS a seguir;5
    E0400 : BOOL ;	//=CH2_2++ZNE02+WIP01;Serviço MES Setpoint não ativo;58
    E0401 : BOOL ;	//=CH2_2++ZNE02+WIP01;Solução para desligamento de linha do MES/PLC para chamada de operadora.;11
    E0402 : BOOL ;	//=CH2_2++ZNE02+WIP01;Serviço MES Tr;10
    E0403 : BOOL ;	//=CH2_2++ZNE02+WIP01;NOK para continuar a partir da estação automática MES (SAService);10
    E0404 : BOOL ;	//=CH2_2++ZNE02+WIP01;Rota Wip do serviço MES não ativa;58
    E0405 : BOOL ;	//=CH2_2++ZNE02+WIP01;Configuração da estação de serviço MES não ativa;58
    E0406 : BOOL ;	//=CH2_2++ZNE02+WIP01;Chamada do Operador de Serviço MES;58
    E0407 : BOOL ;	//=CH2_2++ZNE02+WIP01;Serviço de estação de envio de dados MES SAService não ativo;58
    E0408 : BOOL ;	//=CH2_2++ZNE02+WIP01;Serviço de estação de solicitação de dados MES SRService não ativo;58
    E0409 : BOOL ;	//=CH2_2++ZNE02+WIP01;Serviço de modelo de estação MES SMService não ativo;58
    E0410 : BOOL ;	//=CH2_2++ZNE02+WIP01;Trate wip em modificação;17
    E0411 : BOOL ;	//=CH2_2++ZNE02+WIP01;Estação não automática;16
    E0412 : BOOL ;	//=CH2_2++ZNE02+WIP01;PARADA DE LINHA POR MÊS;17
    E0413 : BOOL ;	//=CH2_2++ZNE02+WIP01;Leitor de bypass CIS NEXT do MES;55
    E0414 : BOOL ;	//=CH2_2++ZNE02+WIP01;Estação excluída;1
    E0415 : BOOL ;	//=CH2_2++ZNE02+WIP01;Lista de estações de configuração de votação;10
    E0416 : BOOL ;
    E0417 : BOOL ;	//=CH2_2++ZNE02+LMN01-DSP01;OPERADOR CHAMADA LIMO 01 ESTAÇÃO 75 SX;53
    E0418 : BOOL ;	//=CH2_2++ZNE02+LMN03-DSP01;OPERADOR CHAMADA LIMO 03 ESTAÇÃO 76 SX;53
    E0419 : BOOL ;	//=CH2_2++ZNE02+LMN05-DSP01;OPERADOR CHAMADA LIMO 05 ESTAÇÃO 77 SX;53
    E0420 : BOOL ;	//=CH2_2++ZNE02+LMN07-DSP01;OPERADOR CHAMADA LIMO 07 ESTAÇÃO 78 SX;53
    E0421 : BOOL ;	//=CH2_2++ZNE02+LMN09-DSP01;OPERADOR CHAMADA LIMO 09 ESTAÇÃO 79 SX;53
    E0422 : BOOL ;	//=CH2_2++ZNE02+LMN11-DSP01;OPERADOR DE LIMO CHAMADA 11 ESTAÇÃO 80 SX;53
    E0423 : BOOL ;	//=CH2_2++ZNE02+LMN13-DSP01;OPERADOR CHAMADA LIMO 13 ESTAÇÃO 81 ESQUERDA;53
    E0424 : BOOL ;	//=CH2_2++ZNE02+LMN15-DSP01;CHAMADA DE OPERADOR DE LIMO 15 ESTAÇÃO Q2 ESQUERDA;53
    E0425 : BOOL ;	//=CH2_2++ZNE02+LMN17-DSP01;CHAMADA DE OPERADOR DE LIMO 17 ESTAÇÃO Q3 ESQUERDA;53
    E0426 : BOOL ;
    E0427 : BOOL ;
    E0428 : BOOL ;
    E0429 : BOOL ;
    E0430 : BOOL ;
    E0431 : BOOL ;
    E0432 : BOOL ;
    E0433 : BOOL ;	//=CH2_2++ZNE02+LMN02-DSP01;OPERADOR CHAMADA LIMO 02 ESTAÇÃO 75 DX;53
    E0434 : BOOL ;	//=CH2_2++ZNE02+LMN04-DSP01;OPERADOR CHAMADA LIMO 04 ESTAÇÃO 76 DX;53
    E0435 : BOOL ;	//=CH2_2++ZNE02+LMN06-DSP01;OPERADOR CHAMADA LIMO 06 ESTAÇÃO 77 DX;53
    E0436 : BOOL ;	//=CH2_2++ZNE02+LMN08-DSP01;OPERADOR CHAMADA LIMO 08 ESTAÇÃO 78 DX;53
    E0437 : BOOL ;	//=CH2_2++ZNE02+LMN10-DSP01;CHAMADA DE OPERADOR LIMO 10 ESTAÇÃO 79 DX;53
    E0438 : BOOL ;	//=CH2_2++ZNE02+LMN12-DSP01;CHAMADA DE OPERADOR LIMO 12 ESTAÇÃO 80 DX;53
    E0439 : BOOL ;	//=CH2_2++ZNE02+LMN14-DSP01;CHAMADA DE OPERADOR LIMO 14 ESTAÇÃO 81 DX;53
    E0440 : BOOL ;	//=CH2_2++ZNE02+LMN16-DSP01;CHAMADA DE OPERADOR DE LIMO 16 ESTAÇÃO Q2 DX;53
    E0441 : BOOL ;	//=CH2_2++ZNE02+LMN18-DSP01;CHAMADA DE OPERADOR DE LIMO 18 ESTAÇÃO Q3 DX;53
    E0442 : BOOL ;
    E0443 : BOOL ;
    E0444 : BOOL ;
    E0445 : BOOL ;
    E0446 : BOOL ;
    E0447 : BOOL ;
    E0448 : BOOL ;
    E0449 : BOOL ;	//=CH2_2++ZNE02+LMN01-DSP01;PARADA LATERAL DO SILT LINE 01 ESTAÇÃO 75 ESQUERDA;12
    E0450 : BOOL ;	//=CH2_2++ZNE02+LMN03-DSP01;PARADA LATERAL DO SILT LINE 03 ESTAÇÃO 76 ESQUERDA;12
    E0451 : BOOL ;	//=CH2_2++ZNE02+LMN05-DSP01;PARADA LATERAL DO SILT LINE 05 ESTAÇÃO 77 ESQUERDA;12
    E0452 : BOOL ;	//=CH2_2++ZNE02+LMN07-DSP01;PARADA LATERAL DO SILT LINE 07 ESTAÇÃO 78 ESQUERDA;12
    E0453 : BOOL ;	//=CH2_2++ZNE02+LMN09-DSP01;PARADA LADO DA LINHA DE LODO 09 ESTAÇÃO 79 ESQUERDA;12
    E0454 : BOOL ;	//=CH2_2++ZNE02+LMN11-DSP01;PARADA LADO DA LINHA DE SILT 11 ESTAÇÃO 80 ESQUERDA;12
    E0455 : BOOL ;	//=CH2_2++ZNE02+LMN13-DSP01;PARADA LADO DA LINHA DE LODO 13 ESTAÇÃO 81 ESQUERDA;12
    E0456 : BOOL ;	//=CH2_2++ZNE02+LMN15-DSP01;PARADA LATERAL DA LINHA DE SILT 15 ESTAÇÃO Q2 ESQUERDA;12
    E0457 : BOOL ;	//=CH2_2++ZNE02+LMN17-DSP01;PARADA LATERAL DO SILT LINE 17 ESTAÇÃO Q3 ESQUERDA;12
    E0458 : BOOL ;
    E0459 : BOOL ;
    E0460 : BOOL ;
    E0461 : BOOL ;
    E0462 : BOOL ;
    E0463 : BOOL ;
    E0464 : BOOL ;
    E0465 : BOOL ;	//=CH2_2++ZNE02+LMN02-DSP01;PARADA LADO DA LINHA DE LODO 02 ESTAÇÃO 75 DIREITA;12
    E0466 : BOOL ;	//=CH2_2++ZNE02+LMN04-DSP01;PARADA LADO DA LINHA DE LODO 04 ESTAÇÃO 76 DIREITA;12
    E0467 : BOOL ;	//=CH2_2++ZNE02+LMN06-DSP01;PARADA LADO DA LINHA DE LODO 06 ESTAÇÃO 77 DIREITA;12
    E0468 : BOOL ;	//=CH2_2++ZNE02+LMN08-DSP01;PARADA LADO DA LINHA DE SILT 08 ESTAÇÃO 78 DIREITA;12
    E0469 : BOOL ;	//=CH2_2++ZNE02+LMN10-DSP01;PARADA LADO DA LINHA DE SILT 10 ESTAÇÃO 79 DIREITA;12
    E0470 : BOOL ;	//=CH2_2++ZNE02+LMN12-DSP01;PARADA LADO DA LINHA DE SILT 12 ESTAÇÃO 80 DIREITA;12
    E0471 : BOOL ;	//=CH2_2++ZNE02+LMN14-DSP01;PARADA LADO DA LINHA DE SILT 14 ESTAÇÃO 81 DIREITA;12
    E0472 : BOOL ;	//=CH2_2++ZNE02+LMN16-DSP01;PARADA LADO DA LINHA DE SILT 16 ESTAÇÃO Q2 DIREITA;12
    E0473 : BOOL ;	//=CH2_2++ZNE02+LMN18-DSP01;PARADA LADO DA LINHA DE SILT 18 ESTAÇÃO Q3 DIREITA;12
    E0474 : BOOL ;
    E0475 : BOOL ;
    E0476 : BOOL ;
    E0477 : BOOL ;
    E0478 : BOOL ;
    E0479 : BOOL ;
    E0480 : BOOL ;
    E0481 : BOOL ;	//=CH2_2++ZNE02+LMN01-DSP01;LINHA PARADA OPERADOR DE LIMO 01 ESTAÇÃO 75 SX;11
    E0482 : BOOL ;	//=CH2_2++ZNE02+LMN03-DSP01;STOP OPERADOR DE LINHA LIMO 03 ESTAÇÃO 76 SX;11
    E0483 : BOOL ;	//=CH2_2++ZNE02+LMN05-DSP01;STOP OPERADOR DE LINHA LIMO 05 ESTAÇÃO 77 SX;11
    E0484 : BOOL ;	//=CH2_2++ZNE02+LMN07-DSP01;PARAR OPERADOR DE LINHA LIMO 07 ESTAÇÃO 78 SX;11
    E0485 : BOOL ;	//=CH2_2++ZNE02+LMN09-DSP01;PARAR OPERADOR DE LINHA LIMO 09 ESTAÇÃO 79 SX;11
    E0486 : BOOL ;	//=CH2_2++ZNE02+LMN11-DSP01;LINE STOP OPERADOR DE LIMO 11 ESTAÇÃO 80 SX;11
    E0487 : BOOL ;	//=CH2_2++ZNE02+LMN13-DSP01;LINHA PARADA OPERADOR DE LIMO 13 ESTAÇÃO 81 ESQUERDA;11
    E0488 : BOOL ;	//=CH2_2++ZNE02+LMN15-DSP01;PARADA DA LINHA DO OPERADOR DE LIMO 15 Q2 ESTAÇÃO À ESQUERDA;11
    E0489 : BOOL ;	//=CH2_2++ZNE02+LMN17-DSP01;PARADA DA LINHA DO OPERADOR DE LIMO 17 Q3 ESTAÇÃO À ESQUERDA;11
    E0490 : BOOL ;
    E0491 : BOOL ;
    E0492 : BOOL ;
    E0493 : BOOL ;
    E0494 : BOOL ;
    E0495 : BOOL ;
    E0496 : BOOL ;
    E0497 : BOOL ;	//=CH2_2++ZNE02+LMN02-DSP01;STOP OPERADOR DE LINHA LIMO 02 ESTAÇÃO 75 DX;11
    E0498 : BOOL ;	//=CH2_2++ZNE02+LMN04-DSP01;STOP OPERADOR DE LINHA LIMO 04 ESTAÇÃO 76 DX;11
    E0499 : BOOL ;	//=CH2_2++ZNE02+LMN06-DSP01;STOP OPERADOR DE LINHA LIMO 06 ESTAÇÃO 77 DX;11
    E0500 : BOOL ;	//=CH2_2++ZNE02+LMN08-DSP01;STOP OPERADOR DE LINHA LIMO 08 ESTAÇÃO 78 DX;11
    E0501 : BOOL ;	//=CH2_2++ZNE02+LMN10-DSP01;STOP LINE OPERADOR LIMO 10 ESTAÇÃO 79 DX;11
    E0502 : BOOL ;	//=CH2_2++ZNE02+LMN12-DSP01;ESTAÇÃO DE PARADA DA LINHA DO OPERADOR LIMO 12 80 DX;11
    E0503 : BOOL ;	//=CH2_2++ZNE02+LMN14-DSP01;PARAR OPERADOR DE LINHA LIMO 14 ESTAÇÃO 81 DX;11
    E0504 : BOOL ;	//=CH2_2++ZNE02+LMN16-DSP01;PARADA DA LINHA DO OPERADOR DE LIMO 16 Q2 ESTAÇÃO DIREITA;11
    E0505 : BOOL ;	//=CH2_2++ZNE02+LMN18-DSP01;PARADA DA LINHA DO OPERADOR DE LIMO 18 Q3 ESTAÇÃO DIREITA;11
    E0506 : BOOL ;
    E0507 : BOOL ;
    E0508 : BOOL ;
    E0509 : BOOL ;
    E0510 : BOOL ;
    E0511 : BOOL ;
    E0512 : BOOL ;
    E0513 : BOOL ;	//=CH2_2++ZNE02+HCZ02-DMC01;FALHA NO MÓDULO ET200S;1
    E0514 : BOOL ;	//=CH2_2++ZNE02+HCZ02-DSW01;FALHA DE SCALANCE;1
    E0515 : BOOL ;	//=CH2_2++ZNE02+HCZ02-QF_06;ALIMENTAÇÃO DISJUNTOR TÉRMICO PARA CIRCUITOS AUXILIARES;1
    E0516 : BOOL ;	//=CH2_2++ZNE02+HCZ02-QF_07;DISJUNTOR TÉRMICO. PODER COMANDOS E SINAIS DE SAÍDA;1
    E0517 : BOOL ;	//=CH2_2++ZNE02+HCZ02-QF_08;FONTE DE ALIMENTAÇÃO MAGNETOTÉRMICA PARA CIRCUITOS DE SEGURANÇA;1
    E0518 : BOOL ;	//=CH2_2++ZNE02+HCZ02-QF_09;DISJUNTOR TÉRMICO. PODER MÓDULOS E SWITCHES E/S ET200;1
    E0519 : BOOL ;
    E0520 : BOOL ;
    E0521 : BOOL ;
    E0522 : BOOL ;
    E0523 : BOOL ;
    E0524 : BOOL ;
    E0525 : BOOL ;
    E0526 : BOOL ;
    E0527 : BOOL ;
    E0528 : BOOL ;
    E0529 : BOOL ;	//=CH2_2++ZNE02+HCZ02-QF_10;ALIMENTAÇÃO 24Vdc MOVIFIT +TQ_01;1
    E0530 : BOOL ;	//=CH2_2++ZNE02+HCZ02-QF_20;FONTE DE ALIMENTAÇÃO 440Vac MOVIFIT +TQ_01;1
    E0531 : BOOL ;	//=CH2_2++ZNE02+HCZ02-QF_21;FONTE DE ALIMENTAÇÃO 440Vac OBTURADOR ENTRADA TTS +TQ_01;1
    E0532 : BOOL ;	//=CH2_2++ZNE02+HCZ02-QF_22;FONTE DE ALIMENTAÇÃO 440Vac SAÍDA TTS DO OBTURADOR +TQ_01;1
    E0533 : BOOL ;	//=CH2_2++ZNE02+HCZ02-QF_25;ALIMENTAÇÃO 440Vac ELEVADOR +TQ_01;1
    E0534 : BOOL ;	//=CH2_2++ZNE02+HCZ02-QF_26;FONTE DE ALIMENTAÇÃO 440Vac ELEVADOR BACKUP +TQ_01;1
    E0535 : BOOL ;	//=CH2_2++ZNE02+HCZ02-QF_27;ALIMENTAÇÃO MAGNETOTÉRMICA 440Vac TRILHA +TTS01;1
    E0536 : BOOL ;	//=CH2_2++ZNE02+HCZ02-QF_30;FONTE DE ALIMENTAÇÃO 440Vac MOTOR FREIO DO ELEVADOR +TQ_01;1
    E0537 : BOOL ;	//=CH2_2++ZNE02+HCZ02-QF_31;FREIO DO MOTOR DE BACKUP DO ELEVADOR 440Vac +TQ_01;1
    E0538 : BOOL ;	//=CH2_2++ZNE02+HCZ02-QF_32;PISTA DE FREIO DO MOTOR DE ALIMENTAÇÃO 440Vac +TTS01;1
    E0539 : BOOL ;	//=CH2_2++ZNE02+HCZ02-BT_01;SOBRETEMP. RESISTOR DE TRAVAGEM DO ELEVADOR +TQ_01;1
    E0540 : BOOL ;	//=CH2_2++ZNE02+HCZ02-BT_02;RESISTÊNCIA À FRENAGEM DO ELEVADOR DE RESERVA.;1
    E0541 : BOOL ;	//=CH2_2++ZNE02+HCZ02-U__01;FALHA MOVIDRIVE +TQ_01;1
    E0542 : BOOL ;	//=CH2_2++ZNE02+HCZ02-U__02;FALHA DE BACKUP DO MOVIDRIVE +TQ_01;1
    E0543 : BOOL ;	//=CH2_2++ZNE02+HCZ02-U__05;FALHA MOVIDRIVE +TTS01;1
    E0544 : BOOL ;	//=CH2_2++ZNE02+HCZ02-U__01;ERRO DE COMUNICAÇÃO MOVIDRIVE +TQ_01;1
    E0545 : BOOL ;	//=CH2_2++ZNE02+HCZ02-U__02;BACKUP MOVIDRIVE +TQ_01 ERRO DE COMUNICAÇÃO;1
    E0546 : BOOL ;	//=CH2_2++ZNE02+HCZ02-U__05;ERRO DE COMUNICAÇÃO MOVIDRIVE +TTS01;1
    E0547 : BOOL ;	//=CH2_2++ZNE02+HCZ02-U__01;EIXO NÃO ZERO MOVIDRIVE +TQ_01;1
    E0548 : BOOL ;	//=CH2_2++ZNE02+HCZ02-U__02;EIXO NÃO ZERO MOVIDRIVE BACKUP +TQ_01;1
    E0549 : BOOL ;	//=CH2_2++ZNE02+HCZ02-KMS02;EFICIÊNCIA DO RELÉ 440Vac +TQ_01;1
    E0550 : BOOL ;	//=CH2_2++ZNE02+HCZ02-KAS02;EFICIÊNCIA DO RELÉ 24Vdc +TQ_01;1
    E0551 : BOOL ;	//=CH2_2++ZNE02+HCZ02-KAS04;FEEDBACK 24Vdc ZONA 2 SETOR 3 TTS01;1
    E0552 : BOOL ;	//=CH2_2++ZNE02+PTZ03-DMC01;FALHA NO MÓDULO ET200S;1
    E0553 : BOOL ;	//=CH2_2++ZNE02+PRE01-DMC01;FALHA NO MÓDULO ET200S;1
    E0554 : BOOL ;	//=CH2_2++ZNE02+XGA03-SC_01;PORTÃO EM ANOMALIA;1
    E0555 : BOOL ;	//=CH2_2++ZNE02+XGA04-SC_01;PORTÃO EM ANOMALIA;1
    E0556 : BOOL ;	//=CH2_2++ZNE02+XGA06-SC_01;PORTÃO EM ANOMALIA;1
    E0557 : BOOL ;	//=CH2_2++ZNE02+XGA07-SC_01;PORTÃO EM ANOMALIA;1
    E0558 : BOOL ;	//=CH2_2++ZNE02+HCZ02-DMC01;ANOMALIA DO MÓDULO ProfSafe ET200S-FDI-FDO;2
    E0559 : BOOL ;
    E0560 : BOOL ;
    E0561 : BOOL ;
    E0562 : BOOL ;
    E0563 : BOOL ;
    E0564 : BOOL ;
    E0565 : BOOL ;
    E0566 : BOOL ;
    E0567 : BOOL ;
    E0568 : BOOL ;
    E0569 : BOOL ;
    E0570 : BOOL ;
    E0571 : BOOL ;
    E0572 : BOOL ;
    E0573 : BOOL ;
    E0574 : BOOL ;
    E0575 : BOOL ;
    E0576 : BOOL ;
    E0577 : BOOL ;
    E0578 : BOOL ;
    E0579 : BOOL ;
    E0580 : BOOL ;
    E0581 : BOOL ;
    E0582 : BOOL ;
    E0583 : BOOL ;
    E0584 : BOOL ;
    E0585 : BOOL ;
    E0586 : BOOL ;
    E0587 : BOOL ;
    E0588 : BOOL ;
    E0589 : BOOL ;
    E0590 : BOOL ;
    E0591 : BOOL ;
    E0592 : BOOL ;
    E0593 : BOOL ;	//=CH2_2++ZNE02+PTZ03-SB_07;BOTÃO DE EMERGENCIA APERTADO;2
    E0594 : BOOL ;	//=CH2_2++ZNE02+PTZ03-SB_07;EMERGÊNCIA NÃO RESTAURADA;2
    E0595 : BOOL ;	//=CH2_2++ZNE02+PRE01-SB_07;BOTÃO DE EMERGENCIA APERTADO;2
    E0596 : BOOL ;	//=CH2_2++ZNE02+PRE01-SB_07;EMERGÊNCIA NÃO RESTAURADA;2
    E0597 : BOOL ;	//=CH2_2++ZNE02+XGA03-SC_01;ACESSO ABERTO NÃO PROGRAMADO (GM);2
    E0598 : BOOL ;	//=CH2_2++ZNE02+XGA03-SC_01;ACESSO NÃO RESTAURADO(GM);2
    E0599 : BOOL ;	//=CH2_2++ZNE02+XGA04-SC_01;ACESSO ABERTO NÃO PROGRAMADO (GM);2
    E0600 : BOOL ;	//=CH2_2++ZNE02+XGA04-SC_01;ACESSO NÃO RESTAURADO(GM);2
    E0601 : BOOL ;	//=CH2_2++ZNE02+PRB05-VT_05;BARREIRA INTERDITADA;2
    E0602 : BOOL ;	//=CH2_2++ZNE02+PRB05-VT_05;BARREIRA NÃO RESTAURADA;2
    E0603 : BOOL ;	//=CH2_2++ZNE02+PGA03-SB_01;BOTÃO DE EMERGENCIA APERTADO;2
    E0604 : BOOL ;	//=CH2_2++ZNE02+PGA03-SB_01;EMERGÊNCIA NÃO RESTAURADA;2
    E0605 : BOOL ;	//=CH2_2++ZNE02+XGA07-SC_01;ACESSO ABERTO NÃO PROGRAMADO (GM);2
    E0606 : BOOL ;	//=CH2_2++ZNE02+XGA07-SC_01;ACESSO NÃO RESTAURADO(GM);2
    E0607 : BOOL ;
    E0608 : BOOL ;
    E0609 : BOOL ;
    E0610 : BOOL ;
    E0611 : BOOL ;
    E0612 : BOOL ;
    E0613 : BOOL ;
    E0614 : BOOL ;
    E0615 : BOOL ;
    E0616 : BOOL ;	//=CH2_2++ZNE02+XGA03-SC_01;ACESSO NÃO RESTAURADO LIMPEZA TÉCNICA (AM);14
    E0617 : BOOL ;	//=CH2_2++ZNE02+XGA03-SC_01;MANUTENÇÃO PROGRAMADA DE ACESSO ABERTO (PM);13
    E0618 : BOOL ;	//=CH2_2++ZNE02+XGA03-SC_01;LIMPEZA TÉCNICA DE ACESSO ABERTO (AM);14
    E0619 : BOOL ;	//=CH2_2++ZNE02+XGA03-SC_01;ACESSO NÃO RESTAURADO PROG. DE MANUTENÇÃO (PM);13
    E0620 : BOOL ;	//=CH2_2++ZNE02+XGA04-SC_01;MANUTENÇÃO PROGRAMADA DE ACESSO ABERTO (PM);13
    E0621 : BOOL ;	//=CH2_2++ZNE02+XGA04-SC_01;LIMPEZA TÉCNICA DE ACESSO ABERTO (AM);14
    E0622 : BOOL ;	//=CH2_2++ZNE02+XGA04-SC_01;ACESSO NÃO RESTAURADO PROG. DE MANUTENÇÃO (PM);13
    E0623 : BOOL ;	//=CH2_2++ZNE02+XGA07-SC_01;MANUTENÇÃO PROGRAMADA DE ACESSO ABERTO (PM);13
    E0624 : BOOL ;	//=CH2_2++ZNE02+XGA07-SC_01;LIMPEZA TÉCNICA DE ACESSO ABERTO (AM);14
    E0625 : BOOL ;	//=CH2_2++ZNE02+XGA07-SC_01;ACESSO NÃO RESTAURADO PROG. DE MANUTENÇÃO (PM);13
    E0626 : BOOL ;	//=CH2_2++ZNE02+XGA04-SC_01;ACESSO NÃO RESTAURADO LIMPEZA TÉCNICA (AM);14
    E0627 : BOOL ;	//=CH2_2++ZNE02+XGA07-SC_01;ACESSO NÃO RESTAURADO LIMPEZA TÉCNICA (AM);14
    E0628 : BOOL ;
    E0629 : BOOL ;
    E0630 : BOOL ;
    E0631 : BOOL ;
    E0632 : BOOL ;
    E0633 : BOOL ;
    E0634 : BOOL ;
    E0635 : BOOL ;
    E0636 : BOOL ;
    E0637 : BOOL ;
    E0638 : BOOL ;
    E0639 : BOOL ;
    E0640 : BOOL ;
    E0641 : BOOL ;	//=CH2_2++ZNE02+HCZ02-QF_03;FONTE DE ALIMENTAÇÃO MAGNETOTÉRMICA PARA AR CONDICIONADO 400V;58
    E0642 : BOOL ;	//=CH2_2++ZNE02+HCZ02-QF_15;MAGNETO. PODER PAINEL OPERADOR 24Vdc +PTZ03;58
    E0643 : BOOL ;	//=CH2_2++ZNE02+HCZ02-QF_16;MAGNETO. PODER PAINEL OPERADOR 24Vdc +PRE01;58
    E0644 : BOOL ;	//=CH2_2++ZNE02+HCZ02-U__01;PRÉ-ALARME MOVIDRIVE +TQ_01;58
    E0645 : BOOL ;	//=CH2_2++ZNE02+HCZ02-U__02;PRÉ-ALARME DE BACKUP DO MOVIDRIVE +TQ_01;58
    E0646 : BOOL ;	//=CH2_2++ZNE02+HCZ02-U__05;PRÉ-ALARME MOVIDRIVE +TTS01;58
    E0647 : BOOL ;	//=CH2_2++ZNE02+PTZ03-DSP01;PRÉ-ALARME SEM PLC <-> COMUNICAÇÃO IHM;58
    E0648 : BOOL ;	//=CH2_2++ZNE02+PRE01-DSP01;PRÉ-ALARME SEM PLC <-> COMUNICAÇÃO IHM;58
    E0649 : BOOL ;	//=CH2_2++ZNE02+PTZ03-SA_03;PEDIDO DE ACESSO PARA MANUTENÇÃO PLANEJADA (PM);58
    E0650 : BOOL ;	//=CH2_2++ZNE02+PTZ03-SA_03;SOLICITAR ACESSO PARA LIMPEZA TÉCNICA (AM);58
    E0651 : BOOL ;	//=CH2_2++ZNE02+PRE01-SA_01;PEDIDO DE ACESSO PARA MANUTENÇÃO PLANEJADA (PM);58
    E0652 : BOOL ;	//=CH2_2++ZNE02+PRE01-SA_03;SOLICITAR ACESSO PARA LIMPEZA TÉCNICA (AM);58
    E0653 : BOOL ;	//=CH2_2++ZNE02+PTZ03-SA_03;SOLICITAR ACESSO PARA LIMPEZA TÉCNICA (AM);58
    E0654 : BOOL ;	//=CH2_2++ZNE02+PRE01-SA_03;SOLICITAR ACESSO PARA MANUTENÇÃO NÃO PROGRAMADA (GM);58
    E0655 : BOOL ;	//=CH2_2++ZNE02+HCZ01-ST_01;CONTROLE DE TEMPERATURA DO GABINETE;58
    E0656 : BOOL ;	//=CH2_2++ZNE02+PTZ03-SA_03;SOLICITAR ACESSO PARA MANUTENÇÃO NÃO PROGRAMADA (GM);58
    E0657 : BOOL ;	//=CH2_2++ZNE02+PGA03-SA_03;SOLICITAR ACESSO PARA MANUTENÇÃO NÃO PROGRAMADA (GM);58
    E0658 : BOOL ;	//=CH2_2++ZNE02+PGA03-SA_03;SOLICITAR ACESSO PARA LIMPEZA TÉCNICA (AM);58
    E0659 : BOOL ;	//=CH2_2++ZNE02+PGA03-SA_03;PEDIDO DE ACESSO PARA MANUTENÇÃO PLANEJADA (PM);58
    E0660 : BOOL ;
    E0661 : BOOL ;
    E0662 : BOOL ;
    E0663 : BOOL ;
    E0664 : BOOL ;
    E0665 : BOOL ;
    E0666 : BOOL ;
    E0667 : BOOL ;
    E0668 : BOOL ;
    E0669 : BOOL ;
    E0670 : BOOL ;
    E0671 : BOOL ;
    E0672 : BOOL ;
    E0673 : BOOL ;	//=CH2_2++ZNE02+WIP01;Desligamento de linha do MES/PLC para chamada da operadora;11
    E0674 : BOOL ;	//=CH2_2++ZNE02+WIP01;Nó do leitor Profinet não está OK;1
    E0675 : BOOL ;	//=CH2_2++ZNE02+WIP01;Placa codificadora de nó Profinet não está OK;1
    E0676 : BOOL ;	//=CH2_2++ZNE02+WIP01;Mau funcionamento do sensor de ritmo;1
    E0677 : BOOL ;	//=CH2_2++ZNE02+WIP01;Disfunção de trânsito de ponto definido;1
    E0678 : BOOL ;	//=CH2_2++ZNE02+WIP01;Mau funcionamento do codificador;1
    E0679 : BOOL ;
    E0680 : BOOL ;
    E0681 : BOOL ;	//=CH2_2++ZNE02+WIP01;Anomalia na leitura de código de barras/etiqueta;5
    E0682 : BOOL ;	//=CH2_2++ZNE02+WIP01;Tempo limite de leitura de código de barras/etiqueta;5
    E0683 : BOOL ;	//=CH2_2++ZNE02+WIP01;Inconsistência físico-lógica;5
    E0684 : BOOL ;	//=CH2_2++ZNE02+WIP01;Dígito de verificação CIS incorreto;5
    E0685 : BOOL ;	//=CH2_2++ZNE02+WIP01;Tempo limite para recepção de dados da rota anterior;5
    E0686 : BOOL ;	//=CH2_2++ZNE02+WIP01;Inconsistência de dados do ponto de ajuste do CIS/VIS com o CIS/VIS a seguir;5
    E0687 : BOOL ;	//=CH2_2++ZNE02+WIP01;Serviço MES Tr;10
    E0688 : BOOL ;	//=CH2_2++ZNE02+WIP01;NOK para continuar a partir da estação automática MES (SAService);10
    E0689 : BOOL ;	//=CH2_2++ZNE02+WIP01;Serviço MES Set Point não ativo;58
    E0690 : BOOL ;	//=CH2_2++ZNE02+WIP01;Rota Wip do serviço MES não ativa;58
    E0691 : BOOL ;	//=CH2_2++ZNE02+WIP01;Configuração da estação de serviço MES não ativa;58
    E0692 : BOOL ;	//=CH2_2++ZNE02+WIP01;Chamada do Operador de Serviço MES;58
    E0693 : BOOL ;	//=CH2_2++ZNE02+WIP01;Serviço de estação de envio de dados MES SAService não ativo;58
    E0694 : BOOL ;	//=CH2_2++ZNE02+WIP01;Serviço de estação de solicitação de dados MES SRService não ativo;10
    E0695 : BOOL ;	//=CH2_2++ZNE02+WIP01;Serviço de modelo de estação MES SMService não ativo;58
    E0696 : BOOL ;
    E0697 : BOOL ;	//=CH2_2++ZNE02+WIP01;Estação não automática;16
    E0698 : BOOL ;	//=CH2_2++ZNE02+WIP01;Leitor de bypass CIS-NEXT da MES;55
    E0699 : BOOL ;	//=CH2_2++ZNE02+WIP01;Estação excluída;17
    E0700 : BOOL ;	//=CH2_2++ZNE02+WIP01;Trate wip em modificação;17
    E0701 : BOOL ;	//=CH2_2++ZNE02+WIP01;Resolvendo Chamada do Operador do MES/PLC (Cogumelo Amarelo);53
    E0702 : BOOL ;
    E0703 : BOOL ;	//=CH2_2++ZNE02+WIP01;Lista de estações de configuração vazia;10
    E0704 : BOOL ;	//=CH2_2++ZNE02+WIP01;Linha Aresto do MES;17
    E0705 : BOOL ;
    E0706 : BOOL ;
    E0707 : BOOL ;
    E0708 : BOOL ;
    E0709 : BOOL ;
    E0710 : BOOL ;
    E0711 : BOOL ;
    E0712 : BOOL ;
    E0713 : BOOL ;
    E0714 : BOOL ;
    E0715 : BOOL ;
    E0716 : BOOL ;
    E0717 : BOOL ;
    E0718 : BOOL ;
    E0719 : BOOL ;
    E0720 : BOOL ;
    E0721 : BOOL ;	//=CH2_2++ZNE02;EM PRODUÇÃO;19
    E0722 : BOOL ;	//=CH2_2++ZNE02+PTZ03-SB_05;INICIAR CICLO AUTOMÁTICO;15
    E0723 : BOOL ;	//=CH2_2++ZNE02+PRE01-SB_05;INICIAR CICLO AUTOMÁTICO;15
    E0724 : BOOL ;	//=CH2_2++ZNE02+PTZ03-SA_01;CICLO MANUAL SELECIONADO;16
    E0725 : BOOL ;	//=CH2_2++ZNE02+PRE01-SA_01;CICLO MANUAL SELECIONADO;16
    E0726 : BOOL ;	//=CH2_2++ZNE02+PTZ03-SB_04;PARADA DO CICLO;17
    E0727 : BOOL ;	//=CH2_2++ZNE02+PRE01-SB_04;PARADA DO CICLO;17
    E0728 : BOOL ;
    E0729 : BOOL ;
    E0730 : BOOL ;
    E0731 : BOOL ;
    E0732 : BOOL ;
    E0733 : BOOL ;
    E0734 : BOOL ;
    E0735 : BOOL ;
    E0736 : BOOL ;
    E0737 : BOOL ;	//=CH2_2++ZNE02+TTS01-SQA01;FALHA NO INTERRUPTOR DE LIMITE DE PARADA;1
    E0738 : BOOL ;	//=CH2_2++ZNE02+TTS01-SQS01;FALHA NO INTERRUPTOR DE LIMITE DE LENTAÇÃO;1
    E0739 : BOOL ;	//=CH2_2++ZNE02+TTS01-SQC01;FALHA NO INTERRUPTOR DE LIMITE DE CONTROLE DE POSIÇÃO;1
    E0740 : BOOL ;	//=CH2_2++ZNE02+TTS01-B__01;FALHA DA FOTOCÉLULA NA PRESENÇA DO VEÍCULO;1
    E0741 : BOOL ;	//=CH2_2++ZNE02+TTS01;SAIR DO TEMPO DE TRANSFERÊNCIA;1
    E0742 : BOOL ;	//=CH2_2++ZNE02+TTS01;CTRL ENGRENAGEM TTS ANTERIOR;1
    E0743 : BOOL ;	//=CH2_2++ZNE02+TTS01;CTRL ENGRENAGEM PRÓXIMO TTS;1
    E0744 : BOOL ;	//=CH2_2++ZNE02+TTS01;POSIÇÃO CTRL;1
    E0745 : BOOL ;	//=CH2_2++ZNE02+TTS01-M__01;FALHA NO INVERSOR;1
    E0746 : BOOL ;	//=CH2_2++ZNE02+TTS01-M__01;ERRO DE COMUNICAÇÃO DO INVERSOR;1
    E0747 : BOOL ;	//=CH2_2++ZNE02+TTS01-SQA02;FALHA DO INTERRUPTOR DE LIMITE DE PROTEÇÃO QUEDA TRABALHO FECHADO;1
    E0748 : BOOL ;	//=CH2_2++ZNE02+TTS01-SQB02;FALHA DE RESTO ABERTO DO INTERRUPTOR DE LIMITE DE PROTEÇÃO QUEDA;1
    E0749 : BOOL ;
    E0750 : BOOL ;	//=CH2_2++ZNE02+TTS01;PRÉ-ALARME DE BYPASS DE FALHA ATIVO;58
    E0751 : BOOL ;	//=CH2_2++ZNE02+TTS01-M__01;PRÉ-ALARME DE CORRENTE ABSORVIDA;58
    E0752 : BOOL ;	//=CH2_2++ZNE02+TTS01-M__01;PRÉ-ALARME DO INVERSOR MOVIMOT;58
    E0753 : BOOL ;	//=CH2_2++ZNE02+TTS01-U__01;ERRO DE COMUNICAÇÃO MOVIFIT;1
    E0754 : BOOL ;	//=CH2_2++ZNE02+TTS01-U__01;INTERRUPTOR MOVIFIT ABERTO 380V;1
    E0755 : BOOL ;	//=CH2_2++ZNE02+TTS01-U__01;AUSÊNCIAS 24 VOLTS MOVIFIT SEGURANÇA;1
    E0756 : BOOL ;	//=CH2_2++ZNE02+TTS01-U__01;AUSÊNCIAS MOVIFIT 24 VOLT;1
    E0757 : BOOL ;	//=CH2_2++ZNE02+TTS01-U__01;ANOMALIA MOVIFIT MOVIFIT;1
    E0758 : BOOL ;	//=CH2_2++ZNE02+TTS01-U__01;SOBRECARGA DE TENSÃO DE SAÍDA 0 MOVIFIT;1
    E0759 : BOOL ;	//=CH2_2++ZNE02+TTS01-U__01;TENSÃO DE SAÍDA DE SOBRECARGA SAÍDA 1 MOVIFIT;1
    E0760 : BOOL ;	//=CH2_2++ZNE02+TTS01-U__01;SOBRECARGA DE TENSÃO DO MOVIFIT NA SAÍDA 2;1
    E0761 : BOOL ;	//=CH2_2++ZNE02+TTS01-U__01;SOBRECARGA DE TENSÃO DE SAÍDA 3 MOVIFIT;1
    E0762 : BOOL ;	//=CH2_2++ZNE02+TTS01-U__01;SOBRECARGA DE TENSÃO DO SENSOR MOVIFIT GRUPO 1;1
    E0763 : BOOL ;	//=CH2_2++ZNE02+TTS01-U__01;SOBRECARGA DE TENSÃO DO SENSOR MOVIFIT GRUPO 2;1
    E0764 : BOOL ;	//=CH2_2++ZNE02+TTS01-U__01;SOBRECARGA DE TENSÃO DO SENSOR MOVIFIT GRUPO 3;1
    E0765 : BOOL ;	//=CH2_2++ZNE02+TTS01-U__01;SOBRECARGA DE TENSÃO DO SENSOR MOVIFIT GRUPO 4;1
    E0766 : BOOL ;	//=CH2_2++ZNE02+TTS01-U__01;ANOMALIA DE HABILITAÇÃO DO INVERSOR;1
    E0767 : BOOL ;
    E0768 : BOOL ;
    E0769 : BOOL ;	//=CH2_2++ZNE02+TQ_01-SQA02;FALHA NO INTERRUPTOR DE LIMITE DE PARADA;1
    E0770 : BOOL ;	//=CH2_2++ZNE02+TQ_01-SQS01;FALHA NO INTERRUPTOR DE LIMITE DE LENTAÇÃO;1
    E0771 : BOOL ;
    E0772 : BOOL ;
    E0773 : BOOL ;	//=CH2_2++ZNE02+TQ_01;SAIR DO TEMPO DE TRANSFERÊNCIA;1
    E0774 : BOOL ;	//=CH2_2++ZNE02+TQ_01;CTRL ENGRENAGEM TTS ANTERIOR;1
    E0775 : BOOL ;	//=CH2_2++ZNE02+TQ_01;CTRL ENGRENAGEM PRÓXIMO TTS;1
    E0776 : BOOL ;	//=CH2_2++ZNE02+TQ_01;POSIÇÃO CTRL;1
    E0777 : BOOL ;	//=CH2_2++ZNE02+TQ_01-U__01;FALHA MOVIFIT FC/30;1
    E0778 : BOOL ;	//=CH2_2++ZNE02+TQ_01-U__01;COMUNICAÇÃO MOVIFIT FC/30;1
    E0779 : BOOL ;	//=CH2_2++ZNE02+TQ_01-SQ_01;FALHA NO INTERRUPTOR DE LIMITE DE PROTEÇÃO CONTRA QUEDA DE SAÍDA TTS;1
    E0780 : BOOL ;	//=CH2_2++ZNE02+TQ_01-SQ_02;FALHA NO INTERRUPTOR DE LIMITE DE PROTEÇÃO CONTRA QUEDA DE ENTRADA TTS;1
    E0781 : BOOL ;
    E0782 : BOOL ;	//=CH2_2++ZNE02+TQ_01;TTS FAULT BYPASS PRÉ-ALARME ATIVO;58
    E0783 : BOOL ;	//=CH2_2++ZNE02+TQ_01-M__04;PRÉ-ALARME DE TRILHA TTS DE CORRENTE ABSORVIDA;58
    E0784 : BOOL ;	//=CH2_2++ZNE02+TQ_01-M__04;PRÉ-ALARME MOVIFIT NA ROTA TTS;58
    E0785 : BOOL ;	//=CH2_2++ZNE02+TQ_01-U__01;ERRO DE COMUNICAÇÃO MOVIFIT;1
    E0786 : BOOL ;	//=CH2_2++ZNE02+TQ_01-U__01;INTERRUPTOR MOVIFIT ABERTO 380V;1
    E0787 : BOOL ;	//=CH2_2++ZNE02+TQ_01-U__01;AUSÊNCIAS 24 VOLTS MOVIFIT SEGURANÇA;1
    E0788 : BOOL ;	//=CH2_2++ZNE02+TQ_01-U__01;AUSÊNCIAS MOVIFIT 24 VOLT;1
    E0789 : BOOL ;	//=CH2_2++ZNE02+TQ_01-U__01;ANOMALIA MOVIFIT;1
    E0790 : BOOL ;	//=CH2_2++ZNE02+TQ_01-U__01;SOBRECARGA DE TENSÃO DE SAÍDA 0 MOVIFIT;1
    E0791 : BOOL ;	//=CH2_2++ZNE02+TQ_01-U__01;TENSÃO DE SAÍDA DE SOBRECARGA SAÍDA 1 MOVIFIT;1
    E0792 : BOOL ;	//=CH2_2++ZNE02+TQ_01-U__01;SOBRECARGA DE TENSÃO DO MOVIFIT NA SAÍDA 2;1
    E0793 : BOOL ;	//=CH2_2++ZNE02+TQ_01-U__01;SOBRECARGA DE TENSÃO DE SAÍDA 3 MOVIFIT;1
    E0794 : BOOL ;	//=CH2_2++ZNE02+TQ_01-U__01;SOBRECARGA DE TENSÃO DO SENSOR MOVIFIT GRUPO 1;1
    E0795 : BOOL ;	//=CH2_2++ZNE02+TQ_01-U__01;SOBRECARGA DE TENSÃO DO SENSOR MOVIFIT GRUPO 2;1
    E0796 : BOOL ;	//=CH2_2++ZNE02+TQ_01-U__01;SOBRECARGA DE TENSÃO DO SENSOR MOVIFIT GRUPO 3;1
    E0797 : BOOL ;	//=CH2_2++ZNE02+TQ_01-U__01;SOBRECARGA DE TENSÃO DO SENSOR MOVIFIT GRUPO 4;1
    E0798 : BOOL ;
    E0799 : BOOL ;
    E0800 : BOOL ;
    E0801 : BOOL ;	//=CH2_2++ZNE02+TQ_01-SQE01;ALTA VIAGEM EXTRA;1
    E0802 : BOOL ;	//=CH2_2++ZNE02+TQ_01-SQE02;BAIXA VIAGEM EXTRA;1
    E0803 : BOOL ;	//=CH2_2++ZNE02+TQ_01-SQC01;FALHA NO INTERRUPTOR DE LIMITE ZERO;1
    E0804 : BOOL ;	//=CH2_2++ZNE02+TQ_01-SQ_01;TRAVA 1 NÃO INSERIDA;1
    E0805 : BOOL ;	//=CH2_2++ZNE02+TQ_01-SQ_02;TRAVA 2 NÃO INSERIDA;1
    E0806 : BOOL ;	//=CH2_2++ZNE02+TQ_01-SQ_03;QUEBRA DA CORREIA;1
    E0807 : BOOL ;	//=CH2_2++ZNE02+TQ_01-SQA01;FALHA FC OBTURADOR DA PARTE MÓVEL DESENGATADO;1
    E0808 : BOOL ;	//=CH2_2++ZNE02+TQ_01-SQB01;FC FALHA PEÇA MÓVEL OBTURADOR INSERIDO;1
    E0809 : BOOL ;	//=CH2_2++ZNE02+TQ_01-SQA03;FALHA FC TTS OBTURADOR DE ENTRADA DESATIVADO;1
    E0810 : BOOL ;	//=CH2_2++ZNE02+TQ_01-SQB03;FALHA FC TTS OBTURADOR DE ENTRADA LIGADO;1
    E0811 : BOOL ;	//=CH2_2++ZNE02+TQ_01-SQA04;FC FALHA TTS OBTURADOR DE SAÍDA DESATIVADO;1
    E0812 : BOOL ;	//=CH2_2++ZNE02+TQ_01-SQB04;GUASTO FC OTTURATORE USCITA TTS INSERITO ;1
    E0813 : BOOL ;	//=CH2_2++ZNE02+TQ_01-B__03;GUASTO FTC PORTELLONE APERTO +TQ_01 ;1
    E0814 : BOOL ;	//=CH2_2++ZNE02+TQ_01-SQB05;BUHL01 NON DISINSERITO ;2
    E0815 : BOOL ;
    E0816 : BOOL ;	//=CH2_2++ZNE02+TQ_01-SQB06;BUHL02 NON DISINSERITO ;2
    E0817 : BOOL ;	//=CH2_2++ZNE02+TQ_01-B__01;FALHA FTC FORA DA ENTRADA + FOLGA TQ_01;1
    E0818 : BOOL ;	//=CH2_2++ZNE02+TQ_01-B__02;FALHA FTC FORA DA SAÍDA +TQ_01;1
    E0819 : BOOL ;	//=CH2_2++ZNE02+TQ_01-SP_01;PRESSÃO DE AR ??INSUFICIENTE DE BUHL;1
    E0820 : BOOL ;
    E0821 : BOOL ;
    E0822 : BOOL ;	//=CH2_2++ZNE02+TQ_01;ANOMALIA DE SELEÇÃO DE LINHA/BACKUP MOVIDRIVE;1
    E0823 : BOOL ;	//=CH2_2++ZNE02+TQ_01-U__01;FALHA DE OTQ DO MOVIFIT;1
    E0824 : BOOL ;	//=CH2_2++ZNE02+TQ_01-U__01;ERRO DE COMUNICAÇÃO MOVIFIT OTQ;1
    E0825 : BOOL ;	//=CH2_2++ZNE02+TQ_01-SQB01;TEMPO LIMITE DE INSERÇÃO DO OBTURADOR DA PEÇA MÓVEL;1
    E0826 : BOOL ;	//=CH2_2++ZNE02+TQ_01-SQA01;TEMPO LIMITE DE DESENGATE DO OBTURADOR DA PARTE MÓVEL;1
    E0827 : BOOL ;	//=CH2_2++ZNE02+TQ_01-SQB03;FC TIMEOUT TTS ENTRADA OBTURADOR LIGADO;1
    E0828 : BOOL ;	//=CH2_2++ZNE02+TQ_01-SQA03;FC TIMEOUT TTS OBTURADOR DE ENTRADA DESATIVADO;1
    E0829 : BOOL ;	//=CH2_2++ZNE02+TQ_01-SQB04;FC TIMEOUT TTS SAÍDA OBTURADOR LIGADO;1
    E0830 : BOOL ;	//=CH2_2++ZNE02+TQ_01-SQA04;FC TIMEOUT SHUTTER TTS SAÍDA DESATIVADA;1
    E0831 : BOOL ;	//=CH2_2++ZNE02+TQ_01-SE_01;TEMPO LIMITE DE POSIÇÃO ALTA;1
    E0832 : BOOL ;	//=CH2_2++ZNE02+TQ_01-SE_01;TIMEOUT POSIZIONE BASSA ;1
    E0833 : BOOL ;	//=CH2_2++ZNE02+TQ_01-U__01;PRÉ-ALARME MOVIFIT INVERSOR OTQ;58
    E0834 : BOOL ;	//=CH2_2++ZNE02+TQ_01-U__01;PRÉ-ALARME DE CORRENTE ABSORVIDA DO INVERSOR OTQ;58
    E0835 : BOOL ;
    E0836 : BOOL ;
    E0837 : BOOL ;
    E0838 : BOOL ;	//=CH2_2++ZNE02+TQ_01;PRÉ-ALARME DE CORREIA LENTA DE POSIÇÃO ALTA +TQ_01;58
    E0839 : BOOL ;	//=CH2_2++ZNE02+TQ_01;PRÉ-ALARME DA CORREIA LENTA POSIÇÃO BAIXA +TQ_01;58
    E0840 : BOOL ;
    E0841 : BOOL ;	//=CH2_2++ZNE02+TQ_01;PRÉ-ALARME DE BYPASS DE FALHA ATIVO;58
    E0842 : BOOL ;
    E0843 : BOOL ;
    E0844 : BOOL ;
    E0845 : BOOL ;
    E0846 : BOOL ;
    E0847 : BOOL ;
    E0848 : BOOL ;
    E0849 : BOOL ;
    E0850 : BOOL ;
    E0851 : BOOL ;
    E0852 : BOOL ;
    E0853 : BOOL ;
    E0854 : BOOL ;
    E0855 : BOOL ;
    E0856 : BOOL ;
    E0857 : BOOL ;	//=CH2_2++ZNE02+TQ_01;CICLO AUTOMÁTICO PASSO A PASSO INICIADO;58
    E0858 : BOOL ;
    E0859 : BOOL ;
    E0860 : BOOL ;
    E0861 : BOOL ;
    E0862 : BOOL ;
    E0863 : BOOL ;
    E0864 : BOOL ;
    E0865 : BOOL ;
    E0866 : BOOL ;
    E0867 : BOOL ;
    E0868 : BOOL ;
    E0869 : BOOL ;
    E0870 : BOOL ;
    E0871 : BOOL ;
    E0872 : BOOL ;
    E0873 : BOOL ;
    E0874 : BOOL ;
    E0875 : BOOL ;
    E0876 : BOOL ;
    E0877 : BOOL ;
    E0878 : BOOL ;
    E0879 : BOOL ;
    E0880 : BOOL ;
    E0881 : BOOL ;
    E0882 : BOOL ;
    E0883 : BOOL ;
    E0884 : BOOL ;
    E0885 : BOOL ;
    E0886 : BOOL ;
    E0887 : BOOL ;
    E0888 : BOOL ;
    E0889 : BOOL ;
    E0890 : BOOL ;
    E0891 : BOOL ;
    E0892 : BOOL ;
    E0893 : BOOL ;
    E0894 : BOOL ;
    E0895 : BOOL ;
    E0896 : BOOL ;
    E0897 : BOOL ;
    E0898 : BOOL ;
    E0899 : BOOL ;
    E0900 : BOOL ;
    E0901 : BOOL ;
    E0902 : BOOL ;
    E0903 : BOOL ;
    E0904 : BOOL ;
    E0905 : BOOL ;
    E0906 : BOOL ;
    E0907 : BOOL ;
    E0908 : BOOL ;
    E0909 : BOOL ;
    E0910 : BOOL ;
    E0911 : BOOL ;
    E0912 : BOOL ;
    E0913 : BOOL ;
    E0914 : BOOL ;
    E0915 : BOOL ;
    E0916 : BOOL ;
    E0917 : BOOL ;
    E0918 : BOOL ;
    E0919 : BOOL ;
    E0920 : BOOL ;
    E0921 : BOOL ;
    E0922 : BOOL ;
    E0923 : BOOL ;
    E0924 : BOOL ;
    E0925 : BOOL ;
    E0926 : BOOL ;
    E0927 : BOOL ;
    E0928 : BOOL ;
    E0929 : BOOL ;
    E0930 : BOOL ;
    E0931 : BOOL ;
    E0932 : BOOL ;
    E0933 : BOOL ;
    E0934 : BOOL ;
    E0935 : BOOL ;
    E0936 : BOOL ;
    E0937 : BOOL ;
    E0938 : BOOL ;
    E0939 : BOOL ;
    E0940 : BOOL ;
    E0941 : BOOL ;
    E0942 : BOOL ;
    E0943 : BOOL ;
    E0944 : BOOL ;
    E0945 : BOOL ;
    E0946 : BOOL ;
    E0947 : BOOL ;
    E0948 : BOOL ;
    E0949 : BOOL ;
    E0950 : BOOL ;
    E0951 : BOOL ;
    E0952 : BOOL ;
    E0953 : BOOL ;
    E0954 : BOOL ;
    E0955 : BOOL ;
    E0956 : BOOL ;
    E0957 : BOOL ;
    E0958 : BOOL ;
    E0959 : BOOL ;
    E0960 : BOOL ;
    E0961 : BOOL ;
    E0962 : BOOL ;
    E0963 : BOOL ;
    E0964 : BOOL ;
    E0965 : BOOL ;
    E0966 : BOOL ;
    E0967 : BOOL ;
    E0968 : BOOL ;
    E0969 : BOOL ;
    E0970 : BOOL ;
    E0971 : BOOL ;
    E0972 : BOOL ;
    E0973 : BOOL ;
    E0974 : BOOL ;
    E0975 : BOOL ;
    E0976 : BOOL ;
    E0977 : BOOL ;
    E0978 : BOOL ;
    E0979 : BOOL ;
    E0980 : BOOL ;
    E0981 : BOOL ;
    E0982 : BOOL ;
    E0983 : BOOL ;
    E0984 : BOOL ;
    E0985 : BOOL ;
    E0986 : BOOL ;
    E0987 : BOOL ;
    E0988 : BOOL ;
    E0989 : BOOL ;
    E0990 : BOOL ;
    E0991 : BOOL ;
    E0992 : BOOL ;
    E0993 : BOOL ;
    E0994 : BOOL ;
    E0995 : BOOL ;
    E0996 : BOOL ;
    E0997 : BOOL ;
    E0998 : BOOL ;
    E0999 : BOOL ;
    E1000 : BOOL ;
    E1001 : BOOL ;
    E1002 : BOOL ;
    E1003 : BOOL ;
    E1004 : BOOL ;
    E1005 : BOOL ;
    E1006 : BOOL ;
    E1007 : BOOL ;
    E1008 : BOOL ;
    E1009 : BOOL ;
    E1010 : BOOL ;
    E1011 : BOOL ;
    E1012 : BOOL ;
    E1013 : BOOL ;
    E1014 : BOOL ;
    E1015 : BOOL ;
    E1016 : BOOL ;
    E1017 : BOOL ;
    E1018 : BOOL ;
    E1019 : BOOL ;
    E1020 : BOOL ;
    E1021 : BOOL ;
    E1022 : BOOL ;
    E1023 : BOOL ;
    E1024 : BOOL ;
   END_STRUCT ;
  END_STRUCT ;
BEGIN
   CM_ID := '=CH2_2';
   STATION_ID := '++ZNE02';
   ELEMENT_ID := '';
   DB_ID := 0;
   PART_IDENTIFICATION := '';
   ACT_CYCLE_TIME := 0;
   COUNT_GOOD := 0;
   COUNT_SCRAP := 0;
   ACCUMULATORS[0] := 0;
   ACCUMULATORS[1] := 0;
   ACCUMULATORS[2] := 0;
   ACCUMULATORS[3] := 0;
   ACCUMULATORS[4] := 0;
   ACCUMULATORS[5] := 0;
   ACCUMULATORS[6] := 0;
   ACCUMULATORS[7] := 0;
   ACCUMULATORS[8] := 0;
   ACCUMULATORS[9] := 0;
   ACCUMULATORS[10] := 0;
   ACCUMULATORS[11] := 0;
   ACCUMULATORS[12] := 0;
   ACCUMULATORS[13] := 0;
   ACCUMULATORS[14] := 0;
   ACCUMULATORS[15] := 0;
   SPARE_01[0] := 0;
   SPARE_01[1] := 0;
   SPARE_01[2] := 0;
   SPARE_01[3] := 0;
   SPARE_01[4] := 0;
   SPARE_01[5] := 0;
   SPARE_01[6] := 0;
   SPARE_01[7] := 0;
   SPARE_01[8] := 0;
   SPARE_01[9] := 0;
   SPARE_01[10] := 0;
   SPARE_01[11] := 0;
   SPARE_01[12] := 0;
   SPARE_01[13] := 0;
   SPARE_01[14] := 0;
   SPARE_01[15] := 0;
   SPARE_01[16] := 0;
   SPARE_01[17] := 0;
   CODE_EVENT[0] := 0;
   CODE_EVENT[1] := 0;
   CODE_EVENT[2] := 0;
   CODE_EVENT[3] := 0;
   CODE_EVENT[4] := 0;
   CODE_EVENT[5] := 0;
   CODE_EVENT[6] := 0;
   CODE_EVENT[7] := 0;
   EVENTS.E0001 := FALSE;
   EVENTS.E0002 := FALSE;
   EVENTS.E0003 := FALSE;
   EVENTS.E0004 := FALSE;
   EVENTS.E0005 := FALSE;
   EVENTS.E0006 := FALSE;
   EVENTS.E0007 := FALSE;
   EVENTS.E0008 := FALSE;
   EVENTS.E0009 := FALSE;
   EVENTS.E0010 := FALSE;
   EVENTS.E0011 := FALSE;
   EVENTS.E0012 := FALSE;
   EVENTS.E0013 := FALSE;
   EVENTS.E0014 := FALSE;
   EVENTS.E0015 := FALSE;
   EVENTS.E0016 := FALSE;
   EVENTS.E0017 := FALSE;
   EVENTS.E0018 := FALSE;
   EVENTS.E0019 := FALSE;
   EVENTS.E0020 := FALSE;
   EVENTS.E0021 := FALSE;
   EVENTS.E0022 := FALSE;
   EVENTS.E0023 := FALSE;
   EVENTS.E0024 := FALSE;
   EVENTS.E0025 := FALSE;
   EVENTS.E0026 := FALSE;
   EVENTS.E0027 := FALSE;
   EVENTS.E0028 := FALSE;
   EVENTS.E0029 := FALSE;
   EVENTS.E0030 := FALSE;
   EVENTS.E0031 := FALSE;
   EVENTS.E0032 := FALSE;
   EVENTS.E0033 := FALSE;
   EVENTS.E0034 := FALSE;
   EVENTS.E0035 := FALSE;
   EVENTS.E0036 := FALSE;
   EVENTS.E0037 := FALSE;
   EVENTS.E0038 := FALSE;
   EVENTS.E0039 := FALSE;
   EVENTS.E0040 := FALSE;
   EVENTS.E0041 := FALSE;
   EVENTS.E0042 := FALSE;
   EVENTS.E0043 := FALSE;
   EVENTS.E0044 := FALSE;
   EVENTS.E0045 := FALSE;
   EVENTS.E0046 := FALSE;
   EVENTS.E0047 := FALSE;
   EVENTS.E0048 := FALSE;
   EVENTS.E0049 := FALSE;
   EVENTS.E0050 := FALSE;
   EVENTS.E0051 := FALSE;
   EVENTS.E0052 := FALSE;
   EVENTS.E0053 := FALSE;
   EVENTS.E0054 := FALSE;
   EVENTS.E0055 := FALSE;
   EVENTS.E0056 := FALSE;
   EVENTS.E0057 := FALSE;
   EVENTS.E0058 := FALSE;
   EVENTS.E0059 := FALSE;
   EVENTS.E0060 := FALSE;
   EVENTS.E0061 := FALSE;
   EVENTS.E0062 := FALSE;
   EVENTS.E0063 := FALSE;
   EVENTS.E0064 := FALSE;
   EVENTS.E0065 := FALSE;
   EVENTS.E0066 := FALSE;
   EVENTS.E0067 := FALSE;
   EVENTS.E0068 := FALSE;
   EVENTS.E0069 := FALSE;
   EVENTS.E0070 := FALSE;
   EVENTS.E0071 := FALSE;
   EVENTS.E0072 := FALSE;
   EVENTS.E0073 := FALSE;
   EVENTS.E0074 := FALSE;
   EVENTS.E0075 := FALSE;
   EVENTS.E0076 := FALSE;
   EVENTS.E0077 := FALSE;
   EVENTS.E0078 := FALSE;
   EVENTS.E0079 := FALSE;
   EVENTS.E0080 := FALSE;
   EVENTS.E0081 := FALSE;
   EVENTS.E0082 := FALSE;
   EVENTS.E0083 := FALSE;
   EVENTS.E0084 := FALSE;
   EVENTS.E0085 := FALSE;
   EVENTS.E0086 := FALSE;
   EVENTS.E0087 := FALSE;
   EVENTS.E0088 := FALSE;
   EVENTS.E0089 := FALSE;
   EVENTS.E0090 := FALSE;
   EVENTS.E0091 := FALSE;
   EVENTS.E0092 := FALSE;
   EVENTS.E0093 := FALSE;
   EVENTS.E0094 := FALSE;
   EVENTS.E0095 := FALSE;
   EVENTS.E0096 := FALSE;
   EVENTS.E0097 := FALSE;
   EVENTS.E0098 := FALSE;
   EVENTS.E0099 := FALSE;
   EVENTS.E0100 := FALSE;
   EVENTS.E0101 := FALSE;
   EVENTS.E0102 := FALSE;
   EVENTS.E0103 := FALSE;
   EVENTS.E0104 := FALSE;
   EVENTS.E0105 := FALSE;
   EVENTS.E0106 := FALSE;
   EVENTS.E0107 := FALSE;
   EVENTS.E0108 := FALSE;
   EVENTS.E0109 := FALSE;
   EVENTS.E0110 := FALSE;
   EVENTS.E0111 := FALSE;
   EVENTS.E0112 := FALSE;
   EVENTS.E0113 := FALSE;
   EVENTS.E0114 := FALSE;
   EVENTS.E0115 := FALSE;
   EVENTS.E0116 := FALSE;
   EVENTS.E0117 := FALSE;
   EVENTS.E0118 := FALSE;
   EVENTS.E0119 := FALSE;
   EVENTS.E0120 := FALSE;
   EVENTS.E0121 := FALSE;
   EVENTS.E0122 := FALSE;
   EVENTS.E0123 := FALSE;
   EVENTS.E0124 := FALSE;
   EVENTS.E0125 := FALSE;
   EVENTS.E0126 := FALSE;
   EVENTS.E0127 := FALSE;
   EVENTS.E0128 := FALSE;
   EVENTS.E0129 := FALSE;
   EVENTS.E0130 := FALSE;
   EVENTS.E0131 := FALSE;
   EVENTS.E0132 := FALSE;
   EVENTS.E0133 := FALSE;
   EVENTS.E0134 := FALSE;
   EVENTS.E0135 := FALSE;
   EVENTS.E0136 := FALSE;
   EVENTS.E0137 := FALSE;
   EVENTS.E0138 := FALSE;
   EVENTS.E0139 := FALSE;
   EVENTS.E0140 := FALSE;
   EVENTS.E0141 := FALSE;
   EVENTS.E0142 := FALSE;
   EVENTS.E0143 := FALSE;
   EVENTS.E0144 := FALSE;
   EVENTS.E0145 := FALSE;
   EVENTS.E0146 := FALSE;
   EVENTS.E0147 := FALSE;
   EVENTS.E0148 := FALSE;
   EVENTS.E0149 := FALSE;
   EVENTS.E0150 := FALSE;
   EVENTS.E0151 := FALSE;
   EVENTS.E0152 := FALSE;
   EVENTS.E0153 := FALSE;
   EVENTS.E0154 := FALSE;
   EVENTS.E0155 := FALSE;
   EVENTS.E0156 := FALSE;
   EVENTS.E0157 := FALSE;
   EVENTS.E0158 := FALSE;
   EVENTS.E0159 := FALSE;
   EVENTS.E0160 := FALSE;
   EVENTS.E0161 := FALSE;
   EVENTS.E0162 := FALSE;
   EVENTS.E0163 := FALSE;
   EVENTS.E0164 := FALSE;
   EVENTS.E0165 := FALSE;
   EVENTS.E0166 := FALSE;
   EVENTS.E0167 := FALSE;
   EVENTS.E0168 := FALSE;
   EVENTS.E0169 := FALSE;
   EVENTS.E0170 := FALSE;
   EVENTS.E0171 := FALSE;
   EVENTS.E0172 := FALSE;
   EVENTS.E0173 := FALSE;
   EVENTS.E0174 := FALSE;
   EVENTS.E0175 := FALSE;
   EVENTS.E0176 := FALSE;
   EVENTS.E0177 := FALSE;
   EVENTS.E0178 := FALSE;
   EVENTS.E0179 := FALSE;
   EVENTS.E0180 := FALSE;
   EVENTS.E0181 := FALSE;
   EVENTS.E0182 := FALSE;
   EVENTS.E0183 := FALSE;
   EVENTS.E0184 := FALSE;
   EVENTS.E0185 := FALSE;
   EVENTS.E0186 := FALSE;
   EVENTS.E0187 := FALSE;
   EVENTS.E0188 := FALSE;
   EVENTS.E0189 := FALSE;
   EVENTS.E0190 := FALSE;
   EVENTS.E0191 := FALSE;
   EVENTS.E0192 := FALSE;
   EVENTS.E0193 := FALSE;
   EVENTS.E0194 := FALSE;
   EVENTS.E0195 := FALSE;
   EVENTS.E0196 := FALSE;
   EVENTS.E0197 := FALSE;
   EVENTS.E0198 := FALSE;
   EVENTS.E0199 := FALSE;
   EVENTS.E0200 := FALSE;
   EVENTS.E0201 := FALSE;
   EVENTS.E0202 := FALSE;
   EVENTS.E0203 := FALSE;
   EVENTS.E0204 := FALSE;
   EVENTS.E0205 := FALSE;
   EVENTS.E0206 := FALSE;
   EVENTS.E0207 := FALSE;
   EVENTS.E0208 := FALSE;
   EVENTS.E0209 := FALSE;
   EVENTS.E0210 := FALSE;
   EVENTS.E0211 := FALSE;
   EVENTS.E0212 := FALSE;
   EVENTS.E0213 := FALSE;
   EVENTS.E0214 := FALSE;
   EVENTS.E0215 := FALSE;
   EVENTS.E0216 := FALSE;
   EVENTS.E0217 := FALSE;
   EVENTS.E0218 := FALSE;
   EVENTS.E0219 := FALSE;
   EVENTS.E0220 := FALSE;
   EVENTS.E0221 := FALSE;
   EVENTS.E0222 := FALSE;
   EVENTS.E0223 := FALSE;
   EVENTS.E0224 := FALSE;
   EVENTS.E0225 := FALSE;
   EVENTS.E0226 := FALSE;
   EVENTS.E0227 := FALSE;
   EVENTS.E0228 := FALSE;
   EVENTS.E0229 := FALSE;
   EVENTS.E0230 := FALSE;
   EVENTS.E0231 := FALSE;
   EVENTS.E0232 := FALSE;
   EVENTS.E0233 := FALSE;
   EVENTS.E0234 := FALSE;
   EVENTS.E0235 := FALSE;
   EVENTS.E0236 := FALSE;
   EVENTS.E0237 := FALSE;
   EVENTS.E0238 := FALSE;
   EVENTS.E0239 := FALSE;
   EVENTS.E0240 := FALSE;
   EVENTS.E0241 := FALSE;
   EVENTS.E0242 := FALSE;
   EVENTS.E0243 := FALSE;
   EVENTS.E0244 := FALSE;
   EVENTS.E0245 := FALSE;
   EVENTS.E0246 := FALSE;
   EVENTS.E0247 := FALSE;
   EVENTS.E0248 := FALSE;
   EVENTS.E0249 := FALSE;
   EVENTS.E0250 := FALSE;
   EVENTS.E0251 := FALSE;
   EVENTS.E0252 := FALSE;
   EVENTS.E0253 := FALSE;
   EVENTS.E0254 := FALSE;
   EVENTS.E0255 := FALSE;
   EVENTS.E0256 := FALSE;
   EVENTS.E0257 := FALSE;
   EVENTS.E0258 := FALSE;
   EVENTS.E0259 := FALSE;
   EVENTS.E0260 := FALSE;
   EVENTS.E0261 := FALSE;
   EVENTS.E0262 := FALSE;
   EVENTS.E0263 := FALSE;
   EVENTS.E0264 := FALSE;
   EVENTS.E0265 := FALSE;
   EVENTS.E0266 := FALSE;
   EVENTS.E0267 := FALSE;
   EVENTS.E0268 := FALSE;
   EVENTS.E0269 := FALSE;
   EVENTS.E0270 := FALSE;
   EVENTS.E0271 := FALSE;
   EVENTS.E0272 := FALSE;
   EVENTS.E0273 := FALSE;
   EVENTS.E0274 := FALSE;
   EVENTS.E0275 := FALSE;
   EVENTS.E0276 := FALSE;
   EVENTS.E0277 := FALSE;
   EVENTS.E0278 := FALSE;
   EVENTS.E0279 := FALSE;
   EVENTS.E0280 := FALSE;
   EVENTS.E0281 := FALSE;
   EVENTS.E0282 := FALSE;
   EVENTS.E0283 := FALSE;
   EVENTS.E0284 := FALSE;
   EVENTS.E0285 := FALSE;
   EVENTS.E0286 := FALSE;
   EVENTS.E0287 := FALSE;
   EVENTS.E0288 := FALSE;
   EVENTS.E0289 := FALSE;
   EVENTS.E0290 := FALSE;
   EVENTS.E0291 := FALSE;
   EVENTS.E0292 := FALSE;
   EVENTS.E0293 := FALSE;
   EVENTS.E0294 := FALSE;
   EVENTS.E0295 := FALSE;
   EVENTS.E0296 := FALSE;
   EVENTS.E0297 := FALSE;
   EVENTS.E0298 := FALSE;
   EVENTS.E0299 := FALSE;
   EVENTS.E0300 := FALSE;
   EVENTS.E0301 := FALSE;
   EVENTS.E0302 := FALSE;
   EVENTS.E0303 := FALSE;
   EVENTS.E0304 := FALSE;
   EVENTS.E0305 := FALSE;
   EVENTS.E0306 := FALSE;
   EVENTS.E0307 := FALSE;
   EVENTS.E0308 := FALSE;
   EVENTS.E0309 := FALSE;
   EVENTS.E0310 := FALSE;
   EVENTS.E0311 := FALSE;
   EVENTS.E0312 := FALSE;
   EVENTS.E0313 := FALSE;
   EVENTS.E0314 := FALSE;
   EVENTS.E0315 := FALSE;
   EVENTS.E0316 := FALSE;
   EVENTS.E0317 := FALSE;
   EVENTS.E0318 := FALSE;
   EVENTS.E0319 := FALSE;
   EVENTS.E0320 := FALSE;
   EVENTS.E0321 := FALSE;
   EVENTS.E0322 := FALSE;
   EVENTS.E0323 := FALSE;
   EVENTS.E0324 := FALSE;
   EVENTS.E0325 := FALSE;
   EVENTS.E0326 := FALSE;
   EVENTS.E0327 := FALSE;
   EVENTS.E0328 := FALSE;
   EVENTS.E0329 := FALSE;
   EVENTS.E0330 := FALSE;
   EVENTS.E0331 := FALSE;
   EVENTS.E0332 := FALSE;
   EVENTS.E0333 := FALSE;
   EVENTS.E0334 := FALSE;
   EVENTS.E0335 := FALSE;
   EVENTS.E0336 := FALSE;
   EVENTS.E0337 := FALSE;
   EVENTS.E0338 := FALSE;
   EVENTS.E0339 := FALSE;
   EVENTS.E0340 := FALSE;
   EVENTS.E0341 := FALSE;
   EVENTS.E0342 := FALSE;
   EVENTS.E0343 := FALSE;
   EVENTS.E0344 := FALSE;
   EVENTS.E0345 := FALSE;
   EVENTS.E0346 := FALSE;
   EVENTS.E0347 := FALSE;
   EVENTS.E0348 := FALSE;
   EVENTS.E0349 := FALSE;
   EVENTS.E0350 := FALSE;
   EVENTS.E0351 := FALSE;
   EVENTS.E0352 := FALSE;
   EVENTS.E0353 := FALSE;
   EVENTS.E0354 := FALSE;
   EVENTS.E0355 := FALSE;
   EVENTS.E0356 := FALSE;
   EVENTS.E0357 := FALSE;
   EVENTS.E0358 := FALSE;
   EVENTS.E0359 := FALSE;
   EVENTS.E0360 := FALSE;
   EVENTS.E0361 := FALSE;
   EVENTS.E0362 := FALSE;
   EVENTS.E0363 := FALSE;
   EVENTS.E0364 := FALSE;
   EVENTS.E0365 := FALSE;
   EVENTS.E0366 := FALSE;
   EVENTS.E0367 := FALSE;
   EVENTS.E0368 := FALSE;
   EVENTS.E0369 := TRUE;
   EVENTS.E0370 := FALSE;
   EVENTS.E0371 := FALSE;
   EVENTS.E0372 := FALSE;
   EVENTS.E0373 := FALSE;
   EVENTS.E0374 := FALSE;
   EVENTS.E0375 := FALSE;
   EVENTS.E0376 := FALSE;
   EVENTS.E0377 := FALSE;
   EVENTS.E0378 := FALSE;
   EVENTS.E0379 := FALSE;
   EVENTS.E0380 := FALSE;
   EVENTS.E0381 := FALSE;
   EVENTS.E0382 := FALSE;
   EVENTS.E0383 := FALSE;
   EVENTS.E0384 := FALSE;
   EVENTS.E0385 := FALSE;
   EVENTS.E0386 := FALSE;
   EVENTS.E0387 := FALSE;
   EVENTS.E0388 := FALSE;
   EVENTS.E0389 := FALSE;
   EVENTS.E0390 := FALSE;
   EVENTS.E0391 := FALSE;
   EVENTS.E0392 := FALSE;
   EVENTS.E0393 := FALSE;
   EVENTS.E0394 := FALSE;
   EVENTS.E0395 := FALSE;
   EVENTS.E0396 := FALSE;
   EVENTS.E0397 := FALSE;
   EVENTS.E0398 := FALSE;
   EVENTS.E0399 := FALSE;
   EVENTS.E0400 := FALSE;
   EVENTS.E0401 := FALSE;
   EVENTS.E0402 := FALSE;
   EVENTS.E0403 := FALSE;
   EVENTS.E0404 := FALSE;
   EVENTS.E0405 := FALSE;
   EVENTS.E0406 := FALSE;
   EVENTS.E0407 := FALSE;
   EVENTS.E0408 := FALSE;
   EVENTS.E0409 := FALSE;
   EVENTS.E0410 := FALSE;
   EVENTS.E0411 := FALSE;
   EVENTS.E0412 := FALSE;
   EVENTS.E0413 := FALSE;
   EVENTS.E0414 := FALSE;
   EVENTS.E0415 := FALSE;
   EVENTS.E0416 := FALSE;
   EVENTS.E0417 := FALSE;
   EVENTS.E0418 := FALSE;
   EVENTS.E0419 := FALSE;
   EVENTS.E0420 := FALSE;
   EVENTS.E0421 := FALSE;
   EVENTS.E0422 := FALSE;
   EVENTS.E0423 := FALSE;
   EVENTS.E0424 := FALSE;
   EVENTS.E0425 := FALSE;
   EVENTS.E0426 := FALSE;
   EVENTS.E0427 := FALSE;
   EVENTS.E0428 := FALSE;
   EVENTS.E0429 := FALSE;
   EVENTS.E0430 := FALSE;
   EVENTS.E0431 := FALSE;
   EVENTS.E0432 := FALSE;
   EVENTS.E0433 := FALSE;
   EVENTS.E0434 := FALSE;
   EVENTS.E0435 := FALSE;
   EVENTS.E0436 := FALSE;
   EVENTS.E0437 := FALSE;
   EVENTS.E0438 := FALSE;
   EVENTS.E0439 := FALSE;
   EVENTS.E0440 := FALSE;
   EVENTS.E0441 := FALSE;
   EVENTS.E0442 := FALSE;
   EVENTS.E0443 := FALSE;
   EVENTS.E0444 := FALSE;
   EVENTS.E0445 := FALSE;
   EVENTS.E0446 := FALSE;
   EVENTS.E0447 := FALSE;
   EVENTS.E0448 := FALSE;
   EVENTS.E0449 := FALSE;
   EVENTS.E0450 := FALSE;
   EVENTS.E0451 := FALSE;
   EVENTS.E0452 := FALSE;
   EVENTS.E0453 := FALSE;
   EVENTS.E0454 := FALSE;
   EVENTS.E0455 := FALSE;
   EVENTS.E0456 := FALSE;
   EVENTS.E0457 := FALSE;
   EVENTS.E0458 := FALSE;
   EVENTS.E0459 := FALSE;
   EVENTS.E0460 := FALSE;
   EVENTS.E0461 := FALSE;
   EVENTS.E0462 := FALSE;
   EVENTS.E0463 := FALSE;
   EVENTS.E0464 := FALSE;
   EVENTS.E0465 := FALSE;
   EVENTS.E0466 := FALSE;
   EVENTS.E0467 := FALSE;
   EVENTS.E0468 := FALSE;
   EVENTS.E0469 := FALSE;
   EVENTS.E0470 := FALSE;
   EVENTS.E0471 := FALSE;
   EVENTS.E0472 := FALSE;
   EVENTS.E0473 := FALSE;
   EVENTS.E0474 := FALSE;
   EVENTS.E0475 := FALSE;
   EVENTS.E0476 := FALSE;
   EVENTS.E0477 := FALSE;
   EVENTS.E0478 := FALSE;
   EVENTS.E0479 := FALSE;
   EVENTS.E0480 := FALSE;
   EVENTS.E0481 := FALSE;
   EVENTS.E0482 := FALSE;
   EVENTS.E0483 := FALSE;
   EVENTS.E0484 := FALSE;
   EVENTS.E0485 := FALSE;
   EVENTS.E0486 := FALSE;
   EVENTS.E0487 := FALSE;
   EVENTS.E0488 := FALSE;
   EVENTS.E0489 := FALSE;
   EVENTS.E0490 := FALSE;
   EVENTS.E0491 := FALSE;
   EVENTS.E0492 := FALSE;
   EVENTS.E0493 := FALSE;
   EVENTS.E0494 := FALSE;
   EVENTS.E0495 := FALSE;
   EVENTS.E0496 := FALSE;
   EVENTS.E0497 := FALSE;
   EVENTS.E0498 := FALSE;
   EVENTS.E0499 := FALSE;
   EVENTS.E0500 := FALSE;
   EVENTS.E0501 := FALSE;
   EVENTS.E0502 := FALSE;
   EVENTS.E0503 := FALSE;
   EVENTS.E0504 := FALSE;
   EVENTS.E0505 := FALSE;
   EVENTS.E0506 := FALSE;
   EVENTS.E0507 := FALSE;
   EVENTS.E0508 := FALSE;
   EVENTS.E0509 := FALSE;
   EVENTS.E0510 := FALSE;
   EVENTS.E0511 := FALSE;
   EVENTS.E0512 := FALSE;
   EVENTS.E0513 := FALSE;
   EVENTS.E0514 := FALSE;
   EVENTS.E0515 := FALSE;
   EVENTS.E0516 := FALSE;
   EVENTS.E0517 := FALSE;
   EVENTS.E0518 := FALSE;
   EVENTS.E0519 := FALSE;
   EVENTS.E0520 := FALSE;
   EVENTS.E0521 := FALSE;
   EVENTS.E0522 := FALSE;
   EVENTS.E0523 := FALSE;
   EVENTS.E0524 := FALSE;
   EVENTS.E0525 := FALSE;
   EVENTS.E0526 := FALSE;
   EVENTS.E0527 := FALSE;
   EVENTS.E0528 := FALSE;
   EVENTS.E0529 := FALSE;
   EVENTS.E0530 := FALSE;
   EVENTS.E0531 := FALSE;
   EVENTS.E0532 := FALSE;
   EVENTS.E0533 := FALSE;
   EVENTS.E0534 := FALSE;
   EVENTS.E0535 := FALSE;
   EVENTS.E0536 := FALSE;
   EVENTS.E0537 := FALSE;
   EVENTS.E0538 := FALSE;
   EVENTS.E0539 := FALSE;
   EVENTS.E0540 := FALSE;
   EVENTS.E0541 := FALSE;
   EVENTS.E0542 := FALSE;
   EVENTS.E0543 := FALSE;
   EVENTS.E0544 := FALSE;
   EVENTS.E0545 := FALSE;
   EVENTS.E0546 := FALSE;
   EVENTS.E0547 := FALSE;
   EVENTS.E0548 := FALSE;
   EVENTS.E0549 := FALSE;
   EVENTS.E0550 := FALSE;
   EVENTS.E0551 := FALSE;
   EVENTS.E0552 := FALSE;
   EVENTS.E0553 := FALSE;
   EVENTS.E0554 := FALSE;
   EVENTS.E0555 := FALSE;
   EVENTS.E0556 := FALSE;
   EVENTS.E0557 := FALSE;
   EVENTS.E0558 := FALSE;
   EVENTS.E0559 := FALSE;
   EVENTS.E0560 := FALSE;
   EVENTS.E0561 := FALSE;
   EVENTS.E0562 := FALSE;
   EVENTS.E0563 := FALSE;
   EVENTS.E0564 := FALSE;
   EVENTS.E0565 := FALSE;
   EVENTS.E0566 := FALSE;
   EVENTS.E0567 := FALSE;
   EVENTS.E0568 := FALSE;
   EVENTS.E0569 := FALSE;
   EVENTS.E0570 := FALSE;
   EVENTS.E0571 := FALSE;
   EVENTS.E0572 := FALSE;
   EVENTS.E0573 := FALSE;
   EVENTS.E0574 := FALSE;
   EVENTS.E0575 := FALSE;
   EVENTS.E0576 := FALSE;
   EVENTS.E0577 := FALSE;
   EVENTS.E0578 := FALSE;
   EVENTS.E0579 := FALSE;
   EVENTS.E0580 := FALSE;
   EVENTS.E0581 := FALSE;
   EVENTS.E0582 := FALSE;
   EVENTS.E0583 := FALSE;
   EVENTS.E0584 := FALSE;
   EVENTS.E0585 := FALSE;
   EVENTS.E0586 := FALSE;
   EVENTS.E0587 := FALSE;
   EVENTS.E0588 := FALSE;
   EVENTS.E0589 := FALSE;
   EVENTS.E0590 := FALSE;
   EVENTS.E0591 := FALSE;
   EVENTS.E0592 := FALSE;
   EVENTS.E0593 := FALSE;
   EVENTS.E0594 := FALSE;
   EVENTS.E0595 := FALSE;
   EVENTS.E0596 := FALSE;
   EVENTS.E0597 := FALSE;
   EVENTS.E0598 := FALSE;
   EVENTS.E0599 := FALSE;
   EVENTS.E0600 := FALSE;
   EVENTS.E0601 := FALSE;
   EVENTS.E0602 := FALSE;
   EVENTS.E0603 := FALSE;
   EVENTS.E0604 := FALSE;
   EVENTS.E0605 := FALSE;
   EVENTS.E0606 := FALSE;
   EVENTS.E0607 := FALSE;
   EVENTS.E0608 := FALSE;
   EVENTS.E0609 := FALSE;
   EVENTS.E0610 := FALSE;
   EVENTS.E0611 := FALSE;
   EVENTS.E0612 := FALSE;
   EVENTS.E0613 := FALSE;
   EVENTS.E0614 := FALSE;
   EVENTS.E0615 := FALSE;
   EVENTS.E0616 := FALSE;
   EVENTS.E0617 := FALSE;
   EVENTS.E0618 := FALSE;
   EVENTS.E0619 := FALSE;
   EVENTS.E0620 := FALSE;
   EVENTS.E0621 := FALSE;
   EVENTS.E0622 := FALSE;
   EVENTS.E0623 := FALSE;
   EVENTS.E0624 := FALSE;
   EVENTS.E0625 := FALSE;
   EVENTS.E0626 := FALSE;
   EVENTS.E0627 := FALSE;
   EVENTS.E0628 := FALSE;
   EVENTS.E0629 := FALSE;
   EVENTS.E0630 := FALSE;
   EVENTS.E0631 := FALSE;
   EVENTS.E0632 := FALSE;
   EVENTS.E0633 := FALSE;
   EVENTS.E0634 := FALSE;
   EVENTS.E0635 := FALSE;
   EVENTS.E0636 := FALSE;
   EVENTS.E0637 := FALSE;
   EVENTS.E0638 := FALSE;
   EVENTS.E0639 := FALSE;
   EVENTS.E0640 := FALSE;
   EVENTS.E0641 := FALSE;
   EVENTS.E0642 := FALSE;
   EVENTS.E0643 := FALSE;
   EVENTS.E0644 := FALSE;
   EVENTS.E0645 := FALSE;
   EVENTS.E0646 := FALSE;
   EVENTS.E0647 := FALSE;
   EVENTS.E0648 := FALSE;
   EVENTS.E0649 := FALSE;
   EVENTS.E0650 := FALSE;
   EVENTS.E0651 := FALSE;
   EVENTS.E0652 := FALSE;
   EVENTS.E0653 := FALSE;
   EVENTS.E0654 := FALSE;
   EVENTS.E0655 := FALSE;
   EVENTS.E0656 := FALSE;
   EVENTS.E0657 := FALSE;
   EVENTS.E0658 := FALSE;
   EVENTS.E0659 := FALSE;
   EVENTS.E0660 := FALSE;
   EVENTS.E0661 := FALSE;
   EVENTS.E0662 := FALSE;
   EVENTS.E0663 := FALSE;
   EVENTS.E0664 := FALSE;
   EVENTS.E0665 := FALSE;
   EVENTS.E0666 := FALSE;
   EVENTS.E0667 := FALSE;
   EVENTS.E0668 := FALSE;
   EVENTS.E0669 := FALSE;
   EVENTS.E0670 := FALSE;
   EVENTS.E0671 := FALSE;
   EVENTS.E0672 := FALSE;
   EVENTS.E0673 := FALSE;
   EVENTS.E0674 := FALSE;
   EVENTS.E0675 := FALSE;
   EVENTS.E0676 := FALSE;
   EVENTS.E0677 := FALSE;
   EVENTS.E0678 := FALSE;
   EVENTS.E0679 := FALSE;
   EVENTS.E0680 := FALSE;
   EVENTS.E0681 := FALSE;
   EVENTS.E0682 := FALSE;
   EVENTS.E0683 := FALSE;
   EVENTS.E0684 := FALSE;
   EVENTS.E0685 := FALSE;
   EVENTS.E0686 := FALSE;
   EVENTS.E0687 := FALSE;
   EVENTS.E0688 := FALSE;
   EVENTS.E0689 := FALSE;
   EVENTS.E0690 := FALSE;
   EVENTS.E0691 := FALSE;
   EVENTS.E0692 := FALSE;
   EVENTS.E0693 := FALSE;
   EVENTS.E0694 := FALSE;
   EVENTS.E0695 := FALSE;
   EVENTS.E0696 := FALSE;
   EVENTS.E0697 := FALSE;
   EVENTS.E0698 := FALSE;
   EVENTS.E0699 := FALSE;
   EVENTS.E0700 := FALSE;
   EVENTS.E0701 := FALSE;
   EVENTS.E0702 := FALSE;
   EVENTS.E0703 := FALSE;
   EVENTS.E0704 := FALSE;
   EVENTS.E0705 := FALSE;
   EVENTS.E0706 := FALSE;
   EVENTS.E0707 := FALSE;
   EVENTS.E0708 := FALSE;
   EVENTS.E0709 := FALSE;
   EVENTS.E0710 := FALSE;
   EVENTS.E0711 := FALSE;
   EVENTS.E0712 := FALSE;
   EVENTS.E0713 := FALSE;
   EVENTS.E0714 := FALSE;
   EVENTS.E0715 := FALSE;
   EVENTS.E0716 := FALSE;
   EVENTS.E0717 := FALSE;
   EVENTS.E0718 := FALSE;
   EVENTS.E0719 := FALSE;
   EVENTS.E0720 := FALSE;
   EVENTS.E0721 := FALSE;
   EVENTS.E0722 := FALSE;
   EVENTS.E0723 := FALSE;
   EVENTS.E0724 := FALSE;
   EVENTS.E0725 := FALSE;
   EVENTS.E0726 := FALSE;
   EVENTS.E0727 := FALSE;
   EVENTS.E0728 := FALSE;
   EVENTS.E0729 := FALSE;
   EVENTS.E0730 := FALSE;
   EVENTS.E0731 := FALSE;
   EVENTS.E0732 := FALSE;
   EVENTS.E0733 := FALSE;
   EVENTS.E0734 := FALSE;
   EVENTS.E0735 := FALSE;
   EVENTS.E0736 := FALSE;
   EVENTS.E0737 := FALSE;
   EVENTS.E0738 := FALSE;
   EVENTS.E0739 := FALSE;
   EVENTS.E0740 := FALSE;
   EVENTS.E0741 := FALSE;
   EVENTS.E0742 := FALSE;
   EVENTS.E0743 := FALSE;
   EVENTS.E0744 := FALSE;
   EVENTS.E0745 := FALSE;
   EVENTS.E0746 := FALSE;
   EVENTS.E0747 := FALSE;
   EVENTS.E0748 := FALSE;
   EVENTS.E0749 := FALSE;
   EVENTS.E0750 := FALSE;
   EVENTS.E0751 := FALSE;
   EVENTS.E0752 := FALSE;
   EVENTS.E0753 := FALSE;
   EVENTS.E0754 := FALSE;
   EVENTS.E0755 := FALSE;
   EVENTS.E0756 := FALSE;
   EVENTS.E0757 := FALSE;
   EVENTS.E0758 := FALSE;
   EVENTS.E0759 := FALSE;
   EVENTS.E0760 := FALSE;
   EVENTS.E0761 := FALSE;
   EVENTS.E0762 := FALSE;
   EVENTS.E0763 := FALSE;
   EVENTS.E0764 := FALSE;
   EVENTS.E0765 := FALSE;
   EVENTS.E0766 := FALSE;
   EVENTS.E0767 := FALSE;
   EVENTS.E0768 := FALSE;
   EVENTS.E0769 := FALSE;
   EVENTS.E0770 := FALSE;
   EVENTS.E0771 := FALSE;
   EVENTS.E0772 := FALSE;
   EVENTS.E0773 := FALSE;
   EVENTS.E0774 := FALSE;
   EVENTS.E0775 := FALSE;
   EVENTS.E0776 := FALSE;
   EVENTS.E0777 := FALSE;
   EVENTS.E0778 := FALSE;
   EVENTS.E0779 := FALSE;
   EVENTS.E0780 := FALSE;
   EVENTS.E0781 := FALSE;
   EVENTS.E0782 := FALSE;
   EVENTS.E0783 := FALSE;
   EVENTS.E0784 := FALSE;
   EVENTS.E0785 := FALSE;
   EVENTS.E0786 := FALSE;
   EVENTS.E0787 := FALSE;
   EVENTS.E0788 := FALSE;
   EVENTS.E0789 := FALSE;
   EVENTS.E0790 := FALSE;
   EVENTS.E0791 := FALSE;
   EVENTS.E0792 := FALSE;
   EVENTS.E0793 := FALSE;
   EVENTS.E0794 := FALSE;
   EVENTS.E0795 := FALSE;
   EVENTS.E0796 := FALSE;
   EVENTS.E0797 := FALSE;
   EVENTS.E0798 := FALSE;
   EVENTS.E0799 := FALSE;
   EVENTS.E0800 := FALSE;
   EVENTS.E0801 := FALSE;
   EVENTS.E0802 := FALSE;
   EVENTS.E0803 := FALSE;
   EVENTS.E0804 := FALSE;
   EVENTS.E0805 := FALSE;
   EVENTS.E0806 := FALSE;
   EVENTS.E0807 := FALSE;
   EVENTS.E0808 := FALSE;
   EVENTS.E0809 := FALSE;
   EVENTS.E0810 := FALSE;
   EVENTS.E0811 := FALSE;
   EVENTS.E0812 := FALSE;
   EVENTS.E0813 := FALSE;
   EVENTS.E0814 := FALSE;
   EVENTS.E0815 := FALSE;
   EVENTS.E0816 := FALSE;
   EVENTS.E0817 := FALSE;
   EVENTS.E0818 := FALSE;
   EVENTS.E0819 := FALSE;
   EVENTS.E0820 := FALSE;
   EVENTS.E0821 := FALSE;
   EVENTS.E0822 := FALSE;
   EVENTS.E0823 := FALSE;
   EVENTS.E0824 := FALSE;
   EVENTS.E0825 := FALSE;
   EVENTS.E0826 := FALSE;
   EVENTS.E0827 := FALSE;
   EVENTS.E0828 := FALSE;
   EVENTS.E0829 := FALSE;
   EVENTS.E0830 := FALSE;
   EVENTS.E0831 := FALSE;
   EVENTS.E0832 := FALSE;
   EVENTS.E0833 := FALSE;
   EVENTS.E0834 := FALSE;
   EVENTS.E0835 := FALSE;
   EVENTS.E0836 := FALSE;
   EVENTS.E0837 := FALSE;
   EVENTS.E0838 := FALSE;
   EVENTS.E0839 := FALSE;
   EVENTS.E0840 := FALSE;
   EVENTS.E0841 := FALSE;
   EVENTS.E0842 := FALSE;
   EVENTS.E0843 := FALSE;
   EVENTS.E0844 := FALSE;
   EVENTS.E0845 := FALSE;
   EVENTS.E0846 := FALSE;
   EVENTS.E0847 := FALSE;
   EVENTS.E0848 := FALSE;
   EVENTS.E0849 := FALSE;
   EVENTS.E0850 := FALSE;
   EVENTS.E0851 := FALSE;
   EVENTS.E0852 := FALSE;
   EVENTS.E0853 := FALSE;
   EVENTS.E0854 := FALSE;
   EVENTS.E0855 := FALSE;
   EVENTS.E0856 := FALSE;
   EVENTS.E0857 := FALSE;
   EVENTS.E0858 := FALSE;
   EVENTS.E0859 := FALSE;
   EVENTS.E0860 := FALSE;
   EVENTS.E0861 := FALSE;
   EVENTS.E0862 := FALSE;
   EVENTS.E0863 := FALSE;
   EVENTS.E0864 := FALSE;
   EVENTS.E0865 := FALSE;
   EVENTS.E0866 := FALSE;
   EVENTS.E0867 := FALSE;
   EVENTS.E0868 := FALSE;
   EVENTS.E0869 := FALSE;
   EVENTS.E0870 := FALSE;
   EVENTS.E0871 := FALSE;
   EVENTS.E0872 := FALSE;
   EVENTS.E0873 := FALSE;
   EVENTS.E0874 := FALSE;
   EVENTS.E0875 := FALSE;
   EVENTS.E0876 := FALSE;
   EVENTS.E0877 := FALSE;
   EVENTS.E0878 := FALSE;
   EVENTS.E0879 := FALSE;
   EVENTS.E0880 := FALSE;
   EVENTS.E0881 := FALSE;
   EVENTS.E0882 := FALSE;
   EVENTS.E0883 := FALSE;
   EVENTS.E0884 := FALSE;
   EVENTS.E0885 := FALSE;
   EVENTS.E0886 := FALSE;
   EVENTS.E0887 := FALSE;
   EVENTS.E0888 := FALSE;
   EVENTS.E0889 := FALSE;
   EVENTS.E0890 := FALSE;
   EVENTS.E0891 := FALSE;
   EVENTS.E0892 := FALSE;
   EVENTS.E0893 := FALSE;
   EVENTS.E0894 := FALSE;
   EVENTS.E0895 := FALSE;
   EVENTS.E0896 := FALSE;
   EVENTS.E0897 := FALSE;
   EVENTS.E0898 := FALSE;
   EVENTS.E0899 := FALSE;
   EVENTS.E0900 := FALSE;
   EVENTS.E0901 := FALSE;
   EVENTS.E0902 := FALSE;
   EVENTS.E0903 := FALSE;
   EVENTS.E0904 := FALSE;
   EVENTS.E0905 := FALSE;
   EVENTS.E0906 := FALSE;
   EVENTS.E0907 := FALSE;
   EVENTS.E0908 := FALSE;
   EVENTS.E0909 := FALSE;
   EVENTS.E0910 := FALSE;
   EVENTS.E0911 := FALSE;
   EVENTS.E0912 := FALSE;
   EVENTS.E0913 := FALSE;
   EVENTS.E0914 := FALSE;
   EVENTS.E0915 := FALSE;
   EVENTS.E0916 := FALSE;
   EVENTS.E0917 := FALSE;
   EVENTS.E0918 := FALSE;
   EVENTS.E0919 := FALSE;
   EVENTS.E0920 := FALSE;
   EVENTS.E0921 := FALSE;
   EVENTS.E0922 := FALSE;
   EVENTS.E0923 := FALSE;
   EVENTS.E0924 := FALSE;
   EVENTS.E0925 := FALSE;
   EVENTS.E0926 := FALSE;
   EVENTS.E0927 := FALSE;
   EVENTS.E0928 := FALSE;
   EVENTS.E0929 := FALSE;
   EVENTS.E0930 := FALSE;
   EVENTS.E0931 := FALSE;
   EVENTS.E0932 := FALSE;
   EVENTS.E0933 := FALSE;
   EVENTS.E0934 := FALSE;
   EVENTS.E0935 := FALSE;
   EVENTS.E0936 := FALSE;
   EVENTS.E0937 := FALSE;
   EVENTS.E0938 := FALSE;
   EVENTS.E0939 := FALSE;
   EVENTS.E0940 := FALSE;
   EVENTS.E0941 := FALSE;
   EVENTS.E0942 := FALSE;
   EVENTS.E0943 := FALSE;
   EVENTS.E0944 := FALSE;
   EVENTS.E0945 := FALSE;
   EVENTS.E0946 := FALSE;
   EVENTS.E0947 := FALSE;
   EVENTS.E0948 := FALSE;
   EVENTS.E0949 := FALSE;
   EVENTS.E0950 := FALSE;
   EVENTS.E0951 := FALSE;
   EVENTS.E0952 := FALSE;
   EVENTS.E0953 := FALSE;
   EVENTS.E0954 := FALSE;
   EVENTS.E0955 := FALSE;
   EVENTS.E0956 := FALSE;
   EVENTS.E0957 := FALSE;
   EVENTS.E0958 := FALSE;
   EVENTS.E0959 := FALSE;
   EVENTS.E0960 := FALSE;
   EVENTS.E0961 := FALSE;
   EVENTS.E0962 := FALSE;
   EVENTS.E0963 := FALSE;
   EVENTS.E0964 := FALSE;
   EVENTS.E0965 := FALSE;
   EVENTS.E0966 := FALSE;
   EVENTS.E0967 := FALSE;
   EVENTS.E0968 := FALSE;
   EVENTS.E0969 := FALSE;
   EVENTS.E0970 := FALSE;
   EVENTS.E0971 := FALSE;
   EVENTS.E0972 := FALSE;
   EVENTS.E0973 := FALSE;
   EVENTS.E0974 := FALSE;
   EVENTS.E0975 := FALSE;
   EVENTS.E0976 := FALSE;
   EVENTS.E0977 := FALSE;
   EVENTS.E0978 := FALSE;
   EVENTS.E0979 := FALSE;
   EVENTS.E0980 := FALSE;
   EVENTS.E0981 := FALSE;
   EVENTS.E0982 := FALSE;
   EVENTS.E0983 := FALSE;
   EVENTS.E0984 := FALSE;
   EVENTS.E0985 := FALSE;
   EVENTS.E0986 := FALSE;
   EVENTS.E0987 := FALSE;
   EVENTS.E0988 := FALSE;
   EVENTS.E0989 := FALSE;
   EVENTS.E0990 := FALSE;
   EVENTS.E0991 := FALSE;
   EVENTS.E0992 := FALSE;
   EVENTS.E0993 := FALSE;
   EVENTS.E0994 := FALSE;
   EVENTS.E0995 := FALSE;
   EVENTS.E0996 := FALSE;
   EVENTS.E0997 := FALSE;
   EVENTS.E0998 := FALSE;
   EVENTS.E0999 := FALSE;
   EVENTS.E1000 := FALSE;
   EVENTS.E1001 := FALSE;
   EVENTS.E1002 := FALSE;
   EVENTS.E1003 := FALSE;
   EVENTS.E1004 := FALSE;
   EVENTS.E1005 := FALSE;
   EVENTS.E1006 := FALSE;
   EVENTS.E1007 := FALSE;
   EVENTS.E1008 := FALSE;
   EVENTS.E1009 := FALSE;
   EVENTS.E1010 := FALSE;
   EVENTS.E1011 := FALSE;
   EVENTS.E1012 := FALSE;
   EVENTS.E1013 := FALSE;
   EVENTS.E1014 := FALSE;
   EVENTS.E1015 := FALSE;
   EVENTS.E1016 := FALSE;
   EVENTS.E1017 := FALSE;
   EVENTS.E1018 := FALSE;
   EVENTS.E1019 := FALSE;
   EVENTS.E1020 := FALSE;
   EVENTS.E1021 := FALSE;
   EVENTS.E1022 := FALSE;
   EVENTS.E1023 := FALSE;
   EVENTS.E1024 := FALSE;
END_DATA_BLOCK
